LIN {X 0,Y 523.995,Z 483.842,A -85,B 0,C 180,E1 -4869.262,E2 -4869.262} C_VEL
LIN {X 0,Y 523.998,Z 483.841,A -85,B 0,C 180,E1 -4871.743,E2 -4871.743} C_VEL
LIN {X 0,Y 523.983,Z 483.844,A -85,B 0,C 180,E1 -4875.053,E2 -4875.053} C_VEL
LIN {X 0,Y 523.956,Z 483.847,A -85,B 0,C 180,E1 -4877.97,E2 -4877.97} C_VEL
LIN {X 0,Y 523.964,Z 483.845,A -85,B 0,C 180,E1 -4880.411,E2 -4880.411} C_VEL
LIN {X 0,Y 523.909,Z 483.852,A -85,B 0,C 180,E1 -4882.894,E2 -4882.894} C_VEL
LIN {X 0,Y 523.947,Z 483.847,A -85,B 0,C 180,E1 -4885.419,E2 -4885.419} C_VEL
LIN {X 0,Y 523.964,Z 483.846,A -85,B 0,C 180,E1 -4888,E2 -4888} C_VEL
LIN {X 0,Y 523.946,Z 483.846,A -85,B 0,C 180,E1 -4890.857,E2 -4890.857} C_VEL
LIN {X 0,Y 523.957,Z 483.847,A -85,B 0,C 180,E1 -4893.736,E2 -4893.736} C_VEL
LIN {X 0,Y 523.917,Z 483.849,A -85,B 0,C 180,E1 -4896.405,E2 -4896.405} C_VEL
LIN {X 0,Y 523.956,Z 483.846,A -85,B 0,C 180,E1 -4899.082,E2 -4899.082} C_VEL
LIN {X 0,Y 523.962,Z 483.845,A -85,B 0,C 180,E1 -4902.119,E2 -4902.119} C_VEL
LIN {X 0,Y 523.953,Z 483.846,A -85,B 0,C 180,E1 -4905.31,E2 -4905.31} C_VEL
LIN {X 0,Y 523.92,Z 483.85,A -85,B 0,C 180,E1 -4906.926,E2 -4906.926} C_VEL
LIN {X 0,Y 523.256,Z 483.934,A -85,B 0,C 180,E1 -4907.567,E2 -4907.567} C_VEL
LIN {X 0,Y 520.42,Z 484.287,A -85,B 0,C 180,E1 -4908.609,E2 -4908.609} C_VEL
LIN {X 0,Y 518.024,Z 484.586,A -85,B 0,C 180,E1 -4909.449,E2 -4909.449} C_VEL
LIN {X 0,Y 516.994,Z 484.714,A -85,B 0,C 180,E1 -4910.096,E2 -4910.096} C_VEL
LIN {X 0,Y 516.909,Z 484.722,A -85,B 0,C 180,E1 -4910.316,E2 -4910.316} C_VEL
LIN {X 0,Y 516.884,Z 484.728,A -85,B 0,C 180,E1 -4913.343,E2 -4913.343} C_VEL
LIN {X 0,Y 516.911,Z 484.723,A -85,B 0,C 180,E1 -4916.122,E2 -4916.122} C_VEL
LIN {X 0,Y 516.893,Z 484.726,A -85,B 0,C 180,E1 -4918.936,E2 -4918.936} C_VEL
LIN {X 0,Y 516.922,Z 484.722,A -85,B 0,C 180,E1 -4921.586,E2 -4921.586} C_VEL
LIN {X 0,Y 516.936,Z 484.721,A -85,B 0,C 180,E1 -4924.212,E2 -4924.212} C_VEL
LIN {X 0,Y 516.875,Z 484.728,A -85,B 0,C 180,E1 -4926.778,E2 -4926.778} C_VEL
LIN {X 0,Y 516.942,Z 484.72,A -85,B 0,C 180,E1 -4929.733,E2 -4929.733} C_VEL
LIN {X 0,Y 516.933,Z 484.719,A -85,B 0,C 180,E1 -4932.597,E2 -4932.597} C_VEL
LIN {X 0,Y 516.947,Z 484.718,A -85,B 0,C 180,E1 -4935.031,E2 -4935.031} C_VEL
LIN {X 0,Y 516.971,Z 484.715,A -85,B 0,C 180,E1 -4938.234,E2 -4938.234} C_VEL
LIN {X 0,Y 516.961,Z 484.717,A -85,B 0,C 180,E1 -4941.4,E2 -4941.4} C_VEL
LIN {X 0,Y 517.016,Z 484.71,A -85,B 0,C 180,E1 -4943.757,E2 -4943.757} C_VEL
LIN {X 0,Y 517.09,Z 484.703,A -85,B 0,C 180,E1 -4947.664,E2 -4947.664} C_VEL
LIN {X 0,Y 517.098,Z 484.699,A -85,B 0,C 180,E1 -4950.779,E2 -4950.779} C_VEL
LIN {X 0,Y 517.003,Z 484.713,A -85,B 0,C 180,E1 -4952.338,E2 -4952.338} C_VEL
LIN {X 0,Y 516.745,Z 484.747,A -85,B 0,C 180,E1 -4954.681,E2 -4954.681} C_VEL
LIN {X 0,Y 516.605,Z 485.864,A -85,B 0,C 180,E1 -4956.248,E2 -4956.248} C_VEL
LIN {X 0,Y 516.544,Z 488.063,A -85,B 0,C 180,E1 -4958.608,E2 -4958.608} C_VEL
LIN {X 0,Y 516.481,Z 491.026,A -85,B 0,C 180,E1 -4961.778,E2 -4961.778} C_VEL
LIN {X 0,Y 516.458,Z 493.998,A -85,B 0,C 180,E1 -4964.984,E2 -4964.984} C_VEL
LIN {X 0,Y 516.325,Z 497.059,A -85,B 0,C 180,E1 -4968.244,E2 -4968.244} C_VEL
LIN {X 0,Y 516.284,Z 499.09,A -85,B 0,C 180,E1 -4970.448,E2 -4970.448} C_VEL
LIN {X 0,Y 520.67,Z 515.911,A -85,B 0,C 180,E1 -4970.996,E2 -4970.996} C_VEL
LIN {X 0,Y 520.325,Z 530.084,A -85,B 0,C 180,E1 -4971.44,E2 -4971.44} C_VEL
LIN {X 0,Y 519.941,Z 544.068,A -85,B 0,C 180,E1 -4972.03,E2 -4972.03} C_VEL
LIN {X 0,Y 519.433,Z 557.792,A -85,B 0,C 180,E1 -4972.767,E2 -4972.767} C_VEL
LIN {X 0,Y 518.868,Z 571.154,A -85,B 0,C 180,E1 -4973.657,E2 -4973.657} C_VEL
LIN {X 0,Y 518.342,Z 584.059,A -85,B 0,C 180,E1 -4974.71,E2 -4974.71} C_VEL
LIN {X 0,Y 517.781,Z 596.388,A -85,B 0,C 180,E1 -4975.926,E2 -4975.926} C_VEL
LIN {X 0,Y 517.395,Z 606.182,A -85,B 0,C 180,E1 -4977.068,E2 -4977.068} C_VEL
LIN {X 0,Y 517.038,Z 615.882,A -85,B 0,C 180,E1 -4978.408,E2 -4978.408} C_VEL
LIN {X 0,Y 516.758,Z 624.427,A -85,B 0,C 180,E1 -4979.823,E2 -4979.823} C_VEL
LIN {X 0,Y 516.533,Z 632.07,A -85,B 0,C 180,E1 -4981.361,E2 -4981.361} C_VEL
LIN {X 0,Y 516.343,Z 638.529,A -85,B 0,C 180,E1 -4982.986,E2 -4982.986} C_VEL
LIN {X 0,Y 516.285,Z 642.897,A -85,B 0,C 180,E1 -4984.397,E2 -4984.397} C_VEL
LIN {X 0,Y 516.177,Z 646.315,A -85,B 0,C 180,E1 -4985.836,E2 -4985.836} C_VEL
LIN {X 0,Y 516.137,Z 648.013,A -85,B 0,C 180,E1 -4986.807,E2 -4986.807} C_VEL
LIN {X 0,Y 516.138,Z 649.321,A -85,B 0,C 180,E1 -4987.836,E2 -4987.836} C_VEL
LIN {X 0,Y 516.128,Z 650.278,A -85,B 0,C 180,E1 -4989.089,E2 -4989.089} C_VEL
LIN {X 0,Y 516.139,Z 650.35,A -85,B 0,C 180,E1 -4990.812,E2 -4990.812} C_VEL
LIN {X 0,Y 516.146,Z 649.734,A -85,B 0,C 180,E1 -4991.851,E2 -4991.851} C_VEL
LIN {X 0,Y 516.173,Z 648.562,A -85,B 0,C 180,E1 -4992.904,E2 -4992.904} C_VEL
LIN {X 0,Y 516.264,Z 645.924,A -85,B 0,C 180,E1 -4994.452,E2 -4994.452} C_VEL
LIN {X 0,Y 516.317,Z 641.557,A -85,B 0,C 180,E1 -4996.172,E2 -4996.172} C_VEL
LIN {X 0,Y 516.429,Z 636.204,A -85,B 0,C 180,E1 -4997.742,E2 -4997.742} C_VEL
LIN {X 0,Y 516.543,Z 629.799,A -85,B 0,C 180,E1 -4999.225,E2 -4999.225} C_VEL
LIN {X 0,Y 516.833,Z 621.343,A -85,B 0,C 180,E1 -5000.813,E2 -5000.813} C_VEL
LIN {X 0,Y 517.202,Z 611.617,A -85,B 0,C 180,E1 -5002.303,E2 -5002.303} C_VEL
LIN {X 0,Y 517.602,Z 600.766,A -85,B 0,C 180,E1 -5003.676,E2 -5003.676} C_VEL
LIN {X 0,Y 518.126,Z 589.032,A -85,B 0,C 180,E1 -5004.915,E2 -5004.915} C_VEL
LIN {X 0,Y 518.638,Z 576.91,A -85,B 0,C 180,E1 -5005.988,E2 -5005.988} C_VEL
LIN {X 0,Y 519.165,Z 563.866,A -85,B 0,C 180,E1 -5006.944,E2 -5006.944} C_VEL
LIN {X 0,Y 519.71,Z 549.92,A -85,B 0,C 180,E1 -5007.77,E2 -5007.77} C_VEL
LIN {X 0,Y 520.223,Z 535.183,A -85,B 0,C 180,E1 -5008.455,E2 -5008.455} C_VEL
LIN {X 0,Y 520.534,Z 520.831,A -85,B 0,C 180,E1 -5008.963,E2 -5008.963} C_VEL
LIN {X 0,Y 520.482,Z 515.011,A -85,B 0,C 180,E1 -5009.128,E2 -5009.128} C_VEL
LIN {X 0,Y 517.023,Z 501.814,A -85,B 0,C 180,E1 -5009.551,E2 -5009.551} C_VEL
LIN {X 0,Y 516.31,Z 499.259,A -85,B 0,C 180,E1 -5009.646,E2 -5009.646} C_VEL
LIN {X 0,Y 516.359,Z 496.719,A -85,B 0,C 180,E1 -5012.434,E2 -5012.434} C_VEL
LIN {X 0,Y 516.419,Z 494.464,A -85,B 0,C 180,E1 -5015.046,E2 -5015.046} C_VEL
LIN {X 0,Y 516.472,Z 492.208,A -85,B 0,C 180,E1 -5017.716,E2 -5017.716} C_VEL
LIN {X 0,Y 516.573,Z 490.1,A -85,B 0,C 180,E1 -5020.115,E2 -5020.115} C_VEL
LIN {X 0,Y 516.622,Z 487.924,A -85,B 0,C 180,E1 -5022.585,E2 -5022.585} C_VEL
LIN {X 0,Y 516.669,Z 485.071,A -85,B 0,C 180,E1 -5025.827,E2 -5025.827} C_VEL
LIN {X 0,Y 516.789,Z 484.742,A -85,B 0,C 180,E1 -5027.432,E2 -5027.432} C_VEL
LIN {X 0,Y 516.904,Z 484.725,A -85,B 0,C 180,E1 -5029.819,E2 -5029.819} C_VEL
LIN {X 0,Y 516.976,Z 484.716,A -85,B 0,C 180,E1 -5032.186,E2 -5032.186} C_VEL
LIN {X 0,Y 517.032,Z 484.704,A -85,B 0,C 180,E1 -5034.54,E2 -5034.54} C_VEL
LIN {X 0,Y 517.081,Z 484.704,A -85,B 0,C 180,E1 -5037.663,E2 -5037.663} C_VEL
LIN {X 0,Y 517.091,Z 484.696,A -85,B 0,C 180,E1 -5040.778,E2 -5040.778} C_VEL
LIN {X 0,Y 517.011,Z 484.71,A -85,B 0,C 180,E1 -5043.117,E2 -5043.117} C_VEL
LIN {X 0,Y 517.007,Z 484.706,A -85,B 0,C 180,E1 -5046.243,E2 -5046.243} C_VEL
LIN {X 0,Y 516.952,Z 484.717,A -85,B 0,C 180,E1 -5049.389,E2 -5049.389} C_VEL
LIN {X 0,Y 516.953,Z 484.713,A -85,B 0,C 180,E1 -5051.81,E2 -5051.81} C_VEL
LIN {X 0,Y 516.94,Z 484.717,A -85,B 0,C 180,E1 -5055.146,E2 -5055.146} C_VEL
LIN {X 0,Y 516.921,Z 484.719,A -85,B 0,C 180,E1 -5058.222,E2 -5058.222} C_VEL
LIN {X 0,Y 516.909,Z 484.723,A -85,B 0,C 180,E1 -5060.701,E2 -5060.701} C_VEL
LIN {X 0,Y 516.907,Z 484.723,A -85,B 0,C 180,E1 -5064.072,E2 -5064.072} C_VEL
LIN {X 0,Y 516.925,Z 484.719,A -85,B 0,C 180,E1 -5066.658,E2 -5066.658} C_VEL
LIN {X 0,Y 516.921,Z 484.72,A -85,B 0,C 180,E1 -5069.527,E2 -5069.527} C_VEL
LIN {X 0,Y 516.897,Z 484.721,A -85,B 0,C 180,E1 -5072.544,E2 -5072.544} C_VEL
LIN {X 0,Y 516.88,Z 484.726,A -85,B 0,C 180,E1 -5075.333,E2 -5075.333} C_VEL
LIN {X 0,Y 516.879,Z 484.725,A -85,B 0,C 180,E1 -5077.943,E2 -5077.943} C_VEL
LIN {X 0,Y 516.883,Z 484.723,A -85,B 0,C 180,E1 -5080.741,E2 -5080.741} C_VEL
LIN {X 0,Y 516.902,Z 484.725,A -85,B 0,C 180,E1 -5082.829,E2 -5082.829} C_VEL
LIN {X 0,Y 516.941,Z 484.824,A -85,B 0,C 180,E1 -5084.85,E2 -5084.85} C_VEL
LIN {X 0,Y 517.947,Z 490.869,A -85,B 0,C 180,E1 -5087.805,E2 -5087.805} C_VEL
LIN {X 0,Y 518.047,Z 495.695,A -85,B 0,C 180,E1 -5089.911,E2 -5089.911} C_VEL
LIN {X 0,Y 517.767,Z 502.856,A -85,B 0,C 180,E1 -5092.828,E2 -5092.828} C_VEL
LIN {X 0,Y 517.6,Z 509.05,A -85,B 0,C 180,E1 -5095.231,E2 -5095.231} C_VEL
LIN {X 0,Y 517.428,Z 517.921,A -85,B 0,C 180,E1 -5098.472,E2 -5098.472} C_VEL
LIN {X 0,Y 517.211,Z 526.908,A -85,B 0,C 180,E1 -5101.602,E2 -5101.602} C_VEL
LIN {X 0,Y 517.044,Z 535.926,A -85,B 0,C 180,E1 -5104.649,E2 -5104.649} C_VEL
LIN {X 0,Y 516.914,Z 545.207,A -85,B 0,C 180,E1 -5107.624,E2 -5107.624} C_VEL
LIN {X 0,Y 516.827,Z 554.056,A -85,B 0,C 180,E1 -5110.384,E2 -5110.384} C_VEL
LIN {X 0,Y 520.741,Z 570.926,A -85,B 0,C 180,E1 -5110.845,E2 -5110.845} C_VEL
LIN {X 0,Y 520.347,Z 586.426,A -85,B 0,C 180,E1 -5111.287,E2 -5111.287} C_VEL
LIN {X 0,Y 519.937,Z 601.506,A -85,B 0,C 180,E1 -5111.887,E2 -5111.887} C_VEL
LIN {X 0,Y 519.531,Z 615.077,A -85,B 0,C 180,E1 -5112.584,E2 -5112.584} C_VEL
LIN {X 0,Y 519.01,Z 627.615,A -85,B 0,C 180,E1 -5113.378,E2 -5113.378} C_VEL
LIN {X 0,Y 518.491,Z 640.647,A -85,B 0,C 180,E1 -5114.382,E2 -5114.382} C_VEL
LIN {X 0,Y 517.981,Z 652.324,A -85,B 0,C 180,E1 -5115.463,E2 -5115.463} C_VEL
LIN {X 0,Y 517.552,Z 663.136,A -85,B 0,C 180,E1 -5116.653,E2 -5116.653} C_VEL
LIN {X 0,Y 517.081,Z 673.797,A -85,B 0,C 180,E1 -5118.057,E2 -5118.057} C_VEL
LIN {X 0,Y 516.89,Z 682.414,A -85,B 0,C 180,E1 -5119.423,E2 -5119.423} C_VEL
LIN {X 0,Y 516.638,Z 688.748,A -85,B 0,C 180,E1 -5120.605,E2 -5120.605} C_VEL
LIN {X 0,Y 516.463,Z 695.699,A -85,B 0,C 180,E1 -5122.179,E2 -5122.179} C_VEL
LIN {X 0,Y 516.356,Z 701.161,A -85,B 0,C 180,E1 -5123.749,E2 -5123.749} C_VEL
LIN {X 0,Y 516.239,Z 705.29,A -85,B 0,C 180,E1 -5125.314,E2 -5125.314} C_VEL
LIN {X 0,Y 516.272,Z 708.184,A -85,B 0,C 180,E1 -5126.878,E2 -5126.878} C_VEL
LIN {X 0,Y 516.189,Z 709.909,A -85,B 0,C 180,E1 -5128.439,E2 -5128.439} C_VEL
LIN {X 0,Y 516.151,Z 710.5,A -85,B 0,C 180,E1 -5130,E2 -5130} C_VEL
LIN {X 0,Y 516.189,Z 709.907,A -85,B 0,C 180,E1 -5131.56,E2 -5131.56} C_VEL
LIN {X 0,Y 516.272,Z 708.181,A -85,B 0,C 180,E1 -5133.121,E2 -5133.121} C_VEL
LIN {X 0,Y 516.238,Z 705.289,A -85,B 0,C 180,E1 -5134.685,E2 -5134.685} C_VEL
LIN {X 0,Y 516.349,Z 701.167,A -85,B 0,C 180,E1 -5136.251,E2 -5136.251} C_VEL
LIN {X 0,Y 516.462,Z 695.703,A -85,B 0,C 180,E1 -5137.821,E2 -5137.821} C_VEL
LIN {X 0,Y 516.637,Z 688.746,A -85,B 0,C 180,E1 -5139.394,E2 -5139.394} C_VEL
LIN {X 0,Y 516.971,Z 680.085,A -85,B 0,C 180,E1 -5140.971,E2 -5140.971} C_VEL
LIN {X 0,Y 517.224,Z 671.026,A -85,B 0,C 180,E1 -5142.337,E2 -5142.337} C_VEL
LIN {X 0,Y 517.633,Z 661.513,A -85,B 0,C 180,E1 -5143.544,E2 -5143.544} C_VEL
LIN {X 0,Y 518.114,Z 649.368,A -85,B 0,C 180,E1 -5144.834,E2 -5144.834} C_VEL
LIN {X 0,Y 518.624,Z 637.232,A -85,B 0,C 180,E1 -5145.906,E2 -5145.906} C_VEL
LIN {X 0,Y 519.093,Z 624.775,A -85,B 0,C 180,E1 -5146.821,E2 -5146.821} C_VEL
LIN {X 0,Y 519.647,Z 611.528,A -85,B 0,C 180,E1 -5147.614,E2 -5147.614} C_VEL
LIN {X 0,Y 520.055,Z 598.266,A -85,B 0,C 180,E1 -5148.255,E2 -5148.255} C_VEL
LIN {X 0,Y 520.479,Z 583.266,A -85,B 0,C 180,E1 -5148.816,E2 -5148.816} C_VEL
LIN {X 0,Y 520.641,Z 570.407,A -85,B 0,C 180,E1 -5149.172,E2 -5149.172} C_VEL
LIN {X 0,Y 516.816,Z 554.06,A -85,B 0,C 180,E1 -5149.622,E2 -5149.622} C_VEL
LIN {X 0,Y 516.973,Z 544.246,A -85,B 0,C 180,E1 -5152.794,E2 -5152.794} C_VEL
LIN {X 0,Y 517.135,Z 535.156,A -85,B 0,C 180,E1 -5155.777,E2 -5155.777} C_VEL
LIN {X 0,Y 517.291,Z 526.189,A -85,B 0,C 180,E1 -5158.835,E2 -5158.835} C_VEL
LIN {X 0,Y 517.499,Z 518.635,A -85,B 0,C 180,E1 -5161.529,E2 -5161.529} C_VEL
LIN {X 0,Y 517.644,Z 511.67,A -85,B 0,C 180,E1 -5164.087,E2 -5164.087} C_VEL
LIN {X 0,Y 517.876,Z 503.58,A -85,B 0,C 180,E1 -5167.176,E2 -5167.176} C_VEL
LIN {X 0,Y 518.18,Z 496.323,A -85,B 0,C 180,E1 -5170.093,E2 -5170.093} C_VEL
LIN {X 0,Y 518.175,Z 492.369,A -85,B 0,C 180,E1 -5171.758,E2 -5171.758} C_VEL
LIN {X 0,Y 517.405,Z 487.511,A -85,B 0,C 180,E1 -5173.953,E2 -5173.953} C_VEL
LIN {X 0,Y 516.928,Z 484.72,A -85,B 0,C 180,E1 -5175.285,E2 -5175.285} C_VEL
LIN {X 0,Y 516.922,Z 484.722,A -85,B 0,C 180,E1 -5178.396,E2 -5178.396} C_VEL
LIN {X 0,Y 516.899,Z 484.725,A -85,B 0,C 180,E1 -5181.286,E2 -5181.286} C_VEL
LIN {X 0,Y 516.883,Z 484.727,A -85,B 0,C 180,E1 -5184.221,E2 -5184.221} C_VEL
LIN {X 0,Y 516.89,Z 484.725,A -85,B 0,C 180,E1 -5187.053,E2 -5187.053} C_VEL
LIN {X 0,Y 516.893,Z 484.726,A -85,B 0,C 180,E1 -5189.797,E2 -5189.797} C_VEL
LIN {X 0,Y 516.921,Z 484.72,A -85,B 0,C 180,E1 -5192.467,E2 -5192.467} C_VEL
LIN {X 0,Y 516.902,Z 484.724,A -85,B 0,C 180,E1 -5195.072,E2 -5195.072} C_VEL
LIN {X 0,Y 516.877,Z 484.727,A -85,B 0,C 180,E1 -5198.462,E2 -5198.462} C_VEL
LIN {X 0,Y 516.896,Z 484.726,A -85,B 0,C 180,E1 -5200.955,E2 -5200.955} C_VEL
LIN {X 0,Y 516.908,Z 484.724,A -85,B 0,C 180,E1 -5203.41,E2 -5203.41} C_VEL
LIN {X 0,Y 516.885,Z 484.727,A -85,B 0,C 180,E1 -5205.834,E2 -5205.834} C_VEL
LIN {X 0,Y 516.993,Z 484.714,A -85,B 0,C 180,E1 -5208.235,E2 -5208.235} C_VEL
LIN {X 0,Y 516.964,Z 484.717,A -85,B 0,C 180,E1 -5211.4,E2 -5211.4} C_VEL
LIN {X 0,Y 517.036,Z 484.705,A -85,B 0,C 180,E1 -5214.54,E2 -5214.54} C_VEL
LIN {X 0,Y 517.076,Z 484.703,A -85,B 0,C 180,E1 -5217.663,E2 -5217.663} C_VEL
LIN {X 0,Y 517.086,Z 484.702,A -85,B 0,C 180,E1 -5220.779,E2 -5220.779} C_VEL
LIN {X 0,Y 517.01,Z 484.711,A -85,B 0,C 180,E1 -5223.117,E2 -5223.117} C_VEL
LIN {X 0,Y 517.007,Z 484.71,A -85,B 0,C 180,E1 -5226.244,E2 -5226.244} C_VEL
LIN {X 0,Y 516.949,Z 484.72,A -85,B 0,C 180,E1 -5229.39,E2 -5229.39} C_VEL
LIN {X 0,Y 516.947,Z 484.719,A -85,B 0,C 180,E1 -5231.811,E2 -5231.811} C_VEL
LIN {X 0,Y 516.934,Z 484.721,A -85,B 0,C 180,E1 -5235.147,E2 -5235.147} C_VEL
LIN {X 0,Y 516.917,Z 484.722,A -85,B 0,C 180,E1 -5238.223,E2 -5238.223} C_VEL
LIN {X 0,Y 516.904,Z 484.724,A -85,B 0,C 180,E1 -5240.702,E2 -5240.702} C_VEL
LIN {X 0,Y 516.903,Z 484.723,A -85,B 0,C 180,E1 -5244.073,E2 -5244.073} C_VEL
LIN {X 0,Y 516.923,Z 484.72,A -85,B 0,C 180,E1 -5246.658,E2 -5246.658} C_VEL
LIN {X 0,Y 516.918,Z 484.723,A -85,B 0,C 180,E1 -5249.528,E2 -5249.528} C_VEL
LIN {X 0,Y 516.895,Z 484.725,A -85,B 0,C 180,E1 -5252.546,E2 -5252.546} C_VEL
LIN {X 0,Y 516.878,Z 484.727,A -85,B 0,C 180,E1 -5255.334,E2 -5255.334} C_VEL
LIN {X 0,Y 516.877,Z 484.729,A -85,B 0,C 180,E1 -5257.945,E2 -5257.945} C_VEL
LIN {X 0,Y 516.913,Z 484.721,A -85,B 0,C 180,E1 -5260.739,E2 -5260.739} C_VEL
LIN {X 0,Y 516.879,Z 484.727,A -85,B 0,C 180,E1 -5263.904,E2 -5263.904} C_VEL
LIN {X 0,Y 516.879,Z 484.726,A -85,B 0,C 180,E1 -5266.108,E2 -5266.108} C_VEL
LIN {X 0,Y 516.903,Z 484.725,A -85,B 0,C 180,E1 -5269.262,E2 -5269.262} C_VEL
LIN {X 0,Y 516.909,Z 484.722,A -85,B 0,C 180,E1 -5270.316,E2 -5270.316} C_VEL
LIN {X 0,Y 516.24,Z 484.806,A -85,B 0,C 180,E1 -5270.966,E2 -5270.966} C_VEL
LIN {X 0,Y 513.383,Z 485.163,A -85,B 0,C 180,E1 -5272.021,E2 -5272.021} C_VEL
LIN {X 0,Y 510.964,Z 485.467,A -85,B 0,C 180,E1 -5272.871,E2 -5272.871} C_VEL
LIN {X 0,Y 509.918,Z 485.596,A -85,B 0,C 180,E1 -5273.527,E2 -5273.527} C_VEL
LIN {X 0,Y 509.829,Z 485.605,A -85,B 0,C 180,E1 -5273.75,E2 -5273.75} C_VEL
LIN {X 0,Y 509.861,Z 485.601,A -85,B 0,C 180,E1 -5276.54,E2 -5276.54} C_VEL
LIN {X 0,Y 509.847,Z 485.604,A -85,B 0,C 180,E1 -5279.335,E2 -5279.335} C_VEL
LIN {X 0,Y 509.897,Z 485.598,A -85,B 0,C 180,E1 -5282.056,E2 -5282.056} C_VEL
LIN {X 0,Y 509.881,Z 485.598,A -85,B 0,C 180,E1 -5284.705,E2 -5284.705} C_VEL
LIN {X 0,Y 509.839,Z 485.604,A -85,B 0,C 180,E1 -5287.456,E2 -5287.456} C_VEL
LIN {X 0,Y 509.92,Z 485.596,A -85,B 0,C 180,E1 -5289.846,E2 -5289.846} C_VEL
LIN {X 0,Y 509.889,Z 485.598,A -85,B 0,C 180,E1 -5293.176,E2 -5293.176} C_VEL
LIN {X 0,Y 509.868,Z 485.602,A -85,B 0,C 180,E1 -5295.635,E2 -5295.635} C_VEL
LIN {X 0,Y 509.917,Z 485.594,A -85,B 0,C 180,E1 -5298.875,E2 -5298.875} C_VEL
LIN {X 0,Y 509.926,Z 485.594,A -85,B 0,C 180,E1 -5302.079,E2 -5302.079} C_VEL
LIN {X 0,Y 509.987,Z 485.585,A -85,B 0,C 180,E1 -5304.465,E2 -5304.465} C_VEL
LIN {X 0,Y 510.061,Z 485.578,A -85,B 0,C 180,E1 -5307.631,E2 -5307.631} C_VEL
LIN {X 0,Y 510.069,Z 485.575,A -85,B 0,C 180,E1 -5310.79,E2 -5310.79} C_VEL
LIN {X 0,Y 509.943,Z 485.592,A -85,B 0,C 180,E1 -5312.37,E2 -5312.37} C_VEL
LIN {X 0,Y 509.702,Z 485.624,A -85,B 0,C 180,E1 -5314.746,E2 -5314.746} C_VEL
LIN {X 0,Y 509.527,Z 485.909,A -85,B 0,C 180,E1 -5315.541,E2 -5315.541} C_VEL
LIN {X 0,Y 509.505,Z 488.136,A -85,B 0,C 180,E1 -5317.929,E2 -5317.929} C_VEL
LIN {X 0,Y 509.419,Z 491.088,A -85,B 0,C 180,E1 -5321.137,E2 -5321.137} C_VEL
LIN {X 0,Y 509.387,Z 494.091,A -85,B 0,C 180,E1 -5324.38,E2 -5324.38} C_VEL
LIN {X 0,Y 509.289,Z 497.265,A -85,B 0,C 180,E1 -5327.79,E2 -5327.79} C_VEL
LIN {X 0,Y 509.245,Z 499.51,A -85,B 0,C 180,E1 -5330.183,E2 -5330.183} C_VEL
LIN {X 0,Y 513.235,Z 514.056,A -85,B 0,C 180,E1 -5330.647,E2 -5330.647} C_VEL
LIN {X 0,Y 513.945,Z 517.527,A -85,B 0,C 180,E1 -5330.774,E2 -5330.774} C_VEL
LIN {X 0,Y 513.583,Z 531.701,A -85,B 0,C 180,E1 -5331.239,E2 -5331.239} C_VEL
LIN {X 0,Y 513.135,Z 545.901,A -85,B 0,C 180,E1 -5331.862,E2 -5331.862} C_VEL
LIN {X 0,Y 512.643,Z 558.776,A -85,B 0,C 180,E1 -5332.573,E2 -5332.573} C_VEL
LIN {X 0,Y 512.032,Z 571.804,A -85,B 0,C 180,E1 -5333.456,E2 -5333.456} C_VEL
LIN {X 0,Y 511.472,Z 584.438,A -85,B 0,C 180,E1 -5334.501,E2 -5334.501} C_VEL
LIN {X 0,Y 510.913,Z 596.247,A -85,B 0,C 180,E1 -5335.677,E2 -5335.677} C_VEL
LIN {X 0,Y 510.384,Z 607.493,A -85,B 0,C 180,E1 -5337.027,E2 -5337.027} C_VEL
LIN {X 0,Y 509.977,Z 617.324,A -85,B 0,C 180,E1 -5338.45,E2 -5338.45} C_VEL
LIN {X 0,Y 509.664,Z 626.083,A -85,B 0,C 180,E1 -5339.991,E2 -5339.991} C_VEL
LIN {X 0,Y 509.459,Z 631.923,A -85,B 0,C 180,E1 -5341.207,E2 -5341.207} C_VEL
LIN {X 0,Y 509.279,Z 637.747,A -85,B 0,C 180,E1 -5342.669,E2 -5342.669} C_VEL
LIN {X 0,Y 509.201,Z 642.294,A -85,B 0,C 180,E1 -5344.093,E2 -5344.093} C_VEL
LIN {X 0,Y 509.092,Z 645.666,A -85,B 0,C 180,E1 -5345.462,E2 -5345.462} C_VEL
LIN {X 0,Y 509.042,Z 648.06,A -85,B 0,C 180,E1 -5346.796,E2 -5346.796} C_VEL
LIN {X 0,Y 509.037,Z 649.874,A -85,B 0,C 180,E1 -5348.41,E2 -5348.41} C_VEL
LIN {X 0,Y 509.028,Z 650.382,A -85,B 0,C 180,E1 -5349.428,E2 -5349.428} C_VEL
LIN {X 0,Y 509.051,Z 650.396,A -85,B 0,C 180,E1 -5350.594,E2 -5350.594} C_VEL
LIN {X 0,Y 509.044,Z 649.806,A -85,B 0,C 180,E1 -5351.794,E2 -5351.794} C_VEL
LIN {X 0,Y 509.103,Z 647.535,A -85,B 0,C 180,E1 -5353.648,E2 -5353.648} C_VEL
LIN {X 0,Y 509.195,Z 644.248,A -85,B 0,C 180,E1 -5355.258,E2 -5355.258} C_VEL
LIN {X 0,Y 509.295,Z 639.231,A -85,B 0,C 180,E1 -5357.001,E2 -5357.001} C_VEL
LIN {X 0,Y 509.38,Z 633.476,A -85,B 0,C 180,E1 -5358.527,E2 -5358.527} C_VEL
LIN {X 0,Y 509.652,Z 626.075,A -85,B 0,C 180,E1 -5360.103,E2 -5360.103} C_VEL
LIN {X 0,Y 509.969,Z 617.151,A -85,B 0,C 180,E1 -5361.672,E2 -5361.672} C_VEL
LIN {X 0,Y 510.371,Z 607.96,A -85,B 0,C 180,E1 -5363.004,E2 -5363.004} C_VEL
LIN {X 0,Y 510.904,Z 596.892,A -85,B 0,C 180,E1 -5364.345,E2 -5364.345} C_VEL
LIN {X 0,Y 511.493,Z 585.133,A -85,B 0,C 180,E1 -5365.528,E2 -5365.528} C_VEL
LIN {X 0,Y 512.029,Z 572.556,A -85,B 0,C 180,E1 -5366.581,E2 -5366.581} C_VEL
LIN {X 0,Y 512.573,Z 560.098,A -85,B 0,C 180,E1 -5367.441,E2 -5367.441} C_VEL
LIN {X 0,Y 513.024,Z 547.804,A -85,B 0,C 180,E1 -5368.14,E2 -5368.14} C_VEL
LIN {X 0,Y 513.533,Z 533.681,A -85,B 0,C 180,E1 -5368.778,E2 -5368.778} C_VEL
LIN {X 0,Y 513.915,Z 519.1,A -85,B 0,C 180,E1 -5369.275,E2 -5369.275} C_VEL
LIN {X 0,Y 513.625,Z 515.708,A -85,B 0,C 180,E1 -5369.384,E2 -5369.384} C_VEL
LIN {X 0,Y 510.164,Z 502.851,A -85,B 0,C 180,E1 -5369.813,E2 -5369.813} C_VEL
LIN {X 0,Y 509.276,Z 499.766,A -85,B 0,C 180,E1 -5369.926,E2 -5369.926} C_VEL
LIN {X 0,Y 509.289,Z 497.11,A -85,B 0,C 180,E1 -5372.91,E2 -5372.91} C_VEL
LIN {X 0,Y 509.377,Z 494.831,A -85,B 0,C 180,E1 -5375.59,E2 -5375.59} C_VEL
LIN {X 0,Y 509.42,Z 492.583,A -85,B 0,C 180,E1 -5378.13,E2 -5378.13} C_VEL
LIN {X 0,Y 509.496,Z 490.376,A -85,B 0,C 180,E1 -5380.667,E2 -5380.667} C_VEL
LIN {X 0,Y 509.544,Z 488.22,A -85,B 0,C 180,E1 -5383.163,E2 -5383.163} C_VEL
LIN {X 0,Y 509.626,Z 486.077,A -85,B 0,C 180,E1 -5385.627,E2 -5385.627} C_VEL
LIN {X 0,Y 509.642,Z 485.631,A -85,B 0,C 180,E1 -5386.442,E2 -5386.442} C_VEL
LIN {X 0,Y 509.89,Z 485.596,A -85,B 0,C 180,E1 -5388.874,E2 -5388.874} C_VEL
LIN {X 0,Y 509.949,Z 485.592,A -85,B 0,C 180,E1 -5392.078,E2 -5392.078} C_VEL
LIN {X 0,Y 509.983,Z 485.583,A -85,B 0,C 180,E1 -5394.464,E2 -5394.464} C_VEL
LIN {X 0,Y 510.052,Z 485.579,A -85,B 0,C 180,E1 -5397.631,E2 -5397.631} C_VEL
LIN {X 0,Y 510.061,Z 485.572,A -85,B 0,C 180,E1 -5400.789,E2 -5400.789} C_VEL
LIN {X 0,Y 509.953,Z 485.59,A -85,B 0,C 180,E1 -5403.16,E2 -5403.16} C_VEL
LIN {X 0,Y 509.975,Z 485.582,A -85,B 0,C 180,E1 -5406.329,E2 -5406.329} C_VEL
LIN {X 0,Y 509.913,Z 485.593,A -85,B 0,C 180,E1 -5408.72,E2 -5408.72} C_VEL
LIN {X 0,Y 509.901,Z 485.591,A -85,B 0,C 180,E1 -5411.931,E2 -5411.931} C_VEL
LIN {X 0,Y 509.889,Z 485.595,A -85,B 0,C 180,E1 -5415.242,E2 -5415.242} C_VEL
LIN {X 0,Y 509.884,Z 485.594,A -85,B 0,C 180,E1 -5418.001,E2 -5418.001} C_VEL
LIN {X 0,Y 509.847,Z 485.599,A -85,B 0,C 180,E1 -5421.002,E2 -5421.002} C_VEL
LIN {X 0,Y 509.833,Z 485.599,A -85,B 0,C 180,E1 -5423.563,E2 -5423.563} C_VEL
LIN {X 0,Y 509.91,Z 485.595,A -85,B 0,C 180,E1 -5426.379,E2 -5426.379} C_VEL
LIN {X 0,Y 509.882,Z 485.595,A -85,B 0,C 180,E1 -5428.844,E2 -5428.844} C_VEL
LIN {X 0,Y 509.824,Z 485.606,A -85,B 0,C 180,E1 -5431.59,E2 -5431.59} C_VEL
LIN {X 0,Y 509.851,Z 485.599,A -85,B 0,C 180,E1 -5434.413,E2 -5434.413} C_VEL
LIN {X 0,Y 509.816,Z 485.607,A -85,B 0,C 180,E1 -5437.341,E2 -5437.341} C_VEL
LIN {X 0,Y 509.836,Z 485.6,A -85,B 0,C 180,E1 -5440.382,E2 -5440.382} C_VEL
LIN {X 0,Y 509.837,Z 485.606,A -85,B 0,C 180,E1 -5443.064,E2 -5443.064} C_VEL
LIN {X 0,Y 509.908,Z 485.723,A -85,B 0,C 180,E1 -5444.531,E2 -5444.531} C_VEL
LIN {X 0,Y 510.962,Z 491.92,A -85,B 0,C 180,E1 -5447.626,E2 -5447.626} C_VEL
LIN {X 0,Y 511.065,Z 496.592,A -85,B 0,C 180,E1 -5449.735,E2 -5449.735} C_VEL
LIN {X 0,Y 510.777,Z 503.839,A -85,B 0,C 180,E1 -5452.742,E2 -5452.742} C_VEL
LIN {X 0,Y 510.548,Z 511.373,A -85,B 0,C 180,E1 -5455.683,E2 -5455.683} C_VEL
LIN {X 0,Y 510.336,Z 520.353,A -85,B 0,C 180,E1 -5458.995,E2 -5458.995} C_VEL
LIN {X 0,Y 510.134,Z 529.12,A -85,B 0,C 180,E1 -5462.069,E2 -5462.069} C_VEL
LIN {X 0,Y 509.98,Z 536.811,A -85,B 0,C 180,E1 -5464.71,E2 -5464.71} C_VEL
LIN {X 0,Y 509.83,Z 546.34,A -85,B 0,C 180,E1 -5467.804,E2 -5467.804} C_VEL
LIN {X 0,Y 509.731,Z 553.417,A -85,B 0,C 180,E1 -5470.089,E2 -5470.089} C_VEL
LIN {X 0,Y 513.96,Z 571.801,A -85,B 0,C 180,E1 -5470.616,E2 -5470.616} C_VEL
LIN {X 0,Y 513.556,Z 587.282,A -85,B 0,C 180,E1 -5471.079,E2 -5471.079} C_VEL
LIN {X 0,Y 513.09,Z 602.081,A -85,B 0,C 180,E1 -5471.688,E2 -5471.688} C_VEL
LIN {X 0,Y 512.615,Z 616.313,A -85,B 0,C 180,E1 -5472.445,E2 -5472.445} C_VEL
LIN {X 0,Y 512.03,Z 630.041,A -85,B 0,C 180,E1 -5473.35,E2 -5473.35} C_VEL
LIN {X 0,Y 511.501,Z 642.796,A -85,B 0,C 180,E1 -5474.374,E2 -5474.374} C_VEL
LIN {X 0,Y 510.962,Z 654.164,A -85,B 0,C 180,E1 -5475.462,E2 -5475.462} C_VEL
LIN {X 0,Y 510.504,Z 664.763,A -85,B 0,C 180,E1 -5476.668,E2 -5476.668} C_VEL
LIN {X 0,Y 510.002,Z 675.013,A -85,B 0,C 180,E1 -5478.07,E2 -5478.07} C_VEL
LIN {X 0,Y 509.818,Z 683.53,A -85,B 0,C 180,E1 -5479.475,E2 -5479.475} C_VEL
LIN {X 0,Y 509.537,Z 690.614,A -85,B 0,C 180,E1 -5480.873,E2 -5480.873} C_VEL
LIN {X 0,Y 509.352,Z 697.182,A -85,B 0,C 180,E1 -5482.468,E2 -5482.468} C_VEL
LIN {X 0,Y 509.294,Z 702.319,A -85,B 0,C 180,E1 -5484.059,E2 -5484.059} C_VEL
LIN {X 0,Y 509.159,Z 705.29,A -85,B 0,C 180,E1 -5485.249,E2 -5485.249} C_VEL
LIN {X 0,Y 509.188,Z 708.183,A -85,B 0,C 180,E1 -5486.835,E2 -5486.835} C_VEL
LIN {X 0,Y 509.109,Z 709.909,A -85,B 0,C 180,E1 -5488.418,E2 -5488.418} C_VEL
LIN {X 0,Y 509.062,Z 710.5,A -85,B 0,C 180,E1 -5490,E2 -5490} C_VEL
LIN {X 0,Y 509.109,Z 709.907,A -85,B 0,C 180,E1 -5491.582,E2 -5491.582} C_VEL
LIN {X 0,Y 509.188,Z 708.18,A -85,B 0,C 180,E1 -5493.164,E2 -5493.164} C_VEL
LIN {X 0,Y 509.158,Z 705.289,A -85,B 0,C 180,E1 -5494.75,E2 -5494.75} C_VEL
LIN {X 0,Y 509.26,Z 701.167,A -85,B 0,C 180,E1 -5496.338,E2 -5496.338} C_VEL
LIN {X 0,Y 509.411,Z 695.703,A -85,B 0,C 180,E1 -5497.929,E2 -5497.929} C_VEL
LIN {X 0,Y 509.56,Z 688.746,A -85,B 0,C 180,E1 -5499.526,E2 -5499.526} C_VEL
LIN {X 0,Y 509.954,Z 680.084,A -85,B 0,C 180,E1 -5501.124,E2 -5501.124} C_VEL
LIN {X 0,Y 510.237,Z 671.026,A -85,B 0,C 180,E1 -5502.509,E2 -5502.509} C_VEL
LIN {X 0,Y 510.656,Z 661.5,A -85,B 0,C 180,E1 -5503.733,E2 -5503.733} C_VEL
LIN {X 0,Y 511.165,Z 649.208,A -85,B 0,C 180,E1 -5505.04,E2 -5505.04} C_VEL
LIN {X 0,Y 511.734,Z 636.679,A -85,B 0,C 180,E1 -5506.147,E2 -5506.147} C_VEL
LIN {X 0,Y 512.334,Z 622.831,A -85,B 0,C 180,E1 -5507.152,E2 -5507.152} C_VEL
LIN {X 0,Y 512.838,Z 609.242,A -85,B 0,C 180,E1 -5507.959,E2 -5507.959} C_VEL
LIN {X 0,Y 513.426,Z 594.727,A -85,B 0,C 180,E1 -5508.638,E2 -5508.638} C_VEL
LIN {X 0,Y 513.8,Z 579.228,A -85,B 0,C 180,E1 -5509.187,E2 -5509.187} C_VEL
LIN {X 0,Y 513.887,Z 571.597,A -85,B 0,C 180,E1 -5509.396,E2 -5509.396} C_VEL
LIN {X 0,Y 509.831,Z 554.538,A -85,B 0,C 180,E1 -5509.884,E2 -5509.884} C_VEL
LIN {X 0,Y 509.733,Z 553.637,A -85,B 0,C 180,E1 -5509.931,E2 -5509.931} C_VEL
LIN {X 0,Y 509.938,Z 543.948,A -85,B 0,C 180,E1 -5513.127,E2 -5513.127} C_VEL
LIN {X 0,Y 510.107,Z 534.071,A -85,B 0,C 180,E1 -5516.423,E2 -5516.423} C_VEL
LIN {X 0,Y 510.294,Z 525.939,A -85,B 0,C 180,E1 -5519.269,E2 -5519.269} C_VEL
LIN {X 0,Y 510.45,Z 518.416,A -85,B 0,C 180,E1 -5522.01,E2 -5522.01} C_VEL
LIN {X 0,Y 510.68,Z 510.909,A -85,B 0,C 180,E1 -5524.827,E2 -5524.827} C_VEL
LIN {X 0,Y 510.969,Z 503.468,A -85,B 0,C 180,E1 -5527.738,E2 -5527.738} C_VEL
LIN {X 0,Y 511.235,Z 497.331,A -85,B 0,C 180,E1 -5530.248,E2 -5530.248} C_VEL
LIN {X 0,Y 511.16,Z 493.135,A -85,B 0,C 180,E1 -5532.059,E2 -5532.059} C_VEL
LIN {X 0,Y 510.214,Z 487.603,A -85,B 0,C 180,E1 -5534.627,E2 -5534.627} C_VEL
LIN {X 0,Y 509.874,Z 485.601,A -85,B 0,C 180,E1 -5535.595,E2 -5535.595} C_VEL
LIN {X 0,Y 509.865,Z 485.602,A -85,B 0,C 180,E1 -5538.576,E2 -5538.576} C_VEL
LIN {X 0,Y 509.848,Z 485.604,A -85,B 0,C 180,E1 -5541.785,E2 -5541.785} C_VEL
LIN {X 0,Y 509.838,Z 485.603,A -85,B 0,C 180,E1 -5544.623,E2 -5544.623} C_VEL
LIN {X 0,Y 509.857,Z 485.604,A -85,B 0,C 180,E1 -5547.481,E2 -5547.481} C_VEL
LIN {X 0,Y 509.872,Z 485.598,A -85,B 0,C 180,E1 -5550.268,E2 -5550.268} C_VEL
LIN {X 0,Y 509.878,Z 485.599,A -85,B 0,C 180,E1 -5552.944,E2 -5552.944} C_VEL
LIN {X 0,Y 509.86,Z 485.602,A -85,B 0,C 180,E1 -5555.574,E2 -5555.574} C_VEL
LIN {X 0,Y 509.812,Z 485.607,A -85,B 0,C 180,E1 -5558.148,E2 -5558.148} C_VEL
LIN {X 0,Y 509.856,Z 485.601,A -85,B 0,C 180,E1 -5560.682,E2 -5560.682} C_VEL
LIN {X 0,Y 509.877,Z 485.601,A -85,B 0,C 180,E1 -5563.175,E2 -5563.175} C_VEL
LIN {X 0,Y 509.854,Z 485.602,A -85,B 0,C 180,E1 -5565.634,E2 -5565.634} C_VEL
LIN {X 0,Y 509.915,Z 485.594,A -85,B 0,C 180,E1 -5568.875,E2 -5568.875} C_VEL
LIN {X 0,Y 509.942,Z 485.59,A -85,B 0,C 180,E1 -5572.079,E2 -5572.079} C_VEL
LIN {X 0,Y 509.985,Z 485.583,A -85,B 0,C 180,E1 -5574.465,E2 -5574.465} C_VEL
LIN {X 0,Y 510.047,Z 485.579,A -85,B 0,C 180,E1 -5577.631,E2 -5577.631} C_VEL
LIN {X 0,Y 510.056,Z 485.577,A -85,B 0,C 180,E1 -5580.79,E2 -5580.79} C_VEL
LIN {X 0,Y 509.953,Z 485.59,A -85,B 0,C 180,E1 -5583.16,E2 -5583.16} C_VEL
LIN {X 0,Y 509.974,Z 485.586,A -85,B 0,C 180,E1 -5586.33,E2 -5586.33} C_VEL
LIN {X 0,Y 509.91,Z 485.594,A -85,B 0,C 180,E1 -5588.721,E2 -5588.721} C_VEL
LIN {X 0,Y 509.895,Z 485.597,A -85,B 0,C 180,E1 -5591.932,E2 -5591.932} C_VEL
LIN {X 0,Y 509.884,Z 485.599,A -85,B 0,C 180,E1 -5595.242,E2 -5595.242} C_VEL
LIN {X 0,Y 509.88,Z 485.6,A -85,B 0,C 180,E1 -5598.002,E2 -5598.002} C_VEL
LIN {X 0,Y 509.842,Z 485.603,A -85,B 0,C 180,E1 -5601.002,E2 -5601.002} C_VEL
LIN {X 0,Y 509.828,Z 485.607,A -85,B 0,C 180,E1 -5603.564,E2 -5603.564} C_VEL
LIN {X 0,Y 509.907,Z 485.594,A -85,B 0,C 180,E1 -5606.38,E2 -5606.38} C_VEL
LIN {X 0,Y 509.879,Z 485.597,A -85,B 0,C 180,E1 -5608.845,E2 -5608.845} C_VEL
LIN {X 0,Y 509.82,Z 485.608,A -85,B 0,C 180,E1 -5611.591,E2 -5611.591} C_VEL
LIN {X 0,Y 509.849,Z 485.603,A -85,B 0,C 180,E1 -5614.414,E2 -5614.414} C_VEL
LIN {X 0,Y 509.814,Z 485.607,A -85,B 0,C 180,E1 -5617.342,E2 -5617.342} C_VEL
LIN {X 0,Y 509.875,Z 485.599,A -85,B 0,C 180,E1 -5620.379,E2 -5620.379} C_VEL
LIN {X 0,Y 509.837,Z 485.604,A -85,B 0,C 180,E1 -5623.065,E2 -5623.065} C_VEL
LIN {X 0,Y 509.828,Z 485.607,A -85,B 0,C 180,E1 -5625.793,E2 -5625.793} C_VEL
LIN {X 0,Y 509.864,Z 485.599,A -85,B 0,C 180,E1 -5628.577,E2 -5628.577} C_VEL
LIN {X 0,Y 509.858,Z 485.602,A -85,B 0,C 180,E1 -5631.664,E2 -5631.664} C_VEL
LIN {X 0,Y 509.829,Z 485.605,A -85,B 0,C 180,E1 -5633.75,E2 -5633.75} C_VEL
LIN {X 0,Y 509.164,Z 485.688,A -85,B 0,C 180,E1 -5634.409,E2 -5634.409} C_VEL
LIN {X 0,Y 506.346,Z 486.04,A -85,B 0,C 180,E1 -5635.481,E2 -5635.481} C_VEL
LIN {X 0,Y 503.953,Z 486.339,A -85,B 0,C 180,E1 -5636.345,E2 -5636.345} C_VEL
LIN {X 0,Y 502.905,Z 486.469,A -85,B 0,C 180,E1 -5637.011,E2 -5637.011} C_VEL
LIN {X 0,Y 502.808,Z 486.479,A -85,B 0,C 180,E1 -5637.237,E2 -5637.237} C_VEL
LIN {X 0,Y 502.816,Z 486.479,A -85,B 0,C 180,E1 -5640.066,E2 -5640.066} C_VEL
LIN {X 0,Y 502.837,Z 486.475,A -85,B 0,C 180,E1 -5642.534,E2 -5642.534} C_VEL
LIN {X 0,Y 502.832,Z 486.477,A -85,B 0,C 180,E1 -5645.299,E2 -5645.299} C_VEL
LIN {X 0,Y 502.788,Z 486.483,A -85,B 0,C 180,E1 -5647.828,E2 -5647.828} C_VEL
LIN {X 0,Y 502.828,Z 486.475,A -85,B 0,C 180,E1 -5650.401,E2 -5650.401} C_VEL
LIN {X 0,Y 502.838,Z 486.474,A -85,B 0,C 180,E1 -5652.933,E2 -5652.933} C_VEL
LIN {X 0,Y 502.849,Z 486.476,A -85,B 0,C 180,E1 -5655.43,E2 -5655.43} C_VEL
LIN {X 0,Y 502.882,Z 486.47,A -85,B 0,C 180,E1 -5658.718,E2 -5658.718} C_VEL
LIN {X 0,Y 502.885,Z 486.472,A -85,B 0,C 180,E1 -5661.967,E2 -5661.967} C_VEL
LIN {X 0,Y 502.943,Z 486.462,A -85,B 0,C 180,E1 -5664.387,E2 -5664.387} C_VEL
LIN {X 0,Y 503.031,Z 486.454,A -85,B 0,C 180,E1 -5667.598,E2 -5667.598} C_VEL
LIN {X 0,Y 503.034,Z 486.452,A -85,B 0,C 180,E1 -5670,E2 -5670} C_VEL
LIN {X 0,Y 502.886,Z 486.471,A -85,B 0,C 180,E1 -5672.403,E2 -5672.403} C_VEL
LIN {X 0,Y 502.658,Z 486.501,A -85,B 0,C 180,E1 -5674.813,E2 -5674.813} C_VEL
LIN {X 0,Y 502.463,Z 486.704,A -85,B 0,C 180,E1 -5675.619,E2 -5675.619} C_VEL
LIN {X 0,Y 502.435,Z 488.917,A -85,B 0,C 180,E1 -5678.041,E2 -5678.041} C_VEL
LIN {X 0,Y 502.389,Z 492.276,A -85,B 0,C 180,E1 -5681.693,E2 -5681.693} C_VEL
LIN {X 0,Y 502.308,Z 495.456,A -85,B 0,C 180,E1 -5685.112,E2 -5685.112} C_VEL
LIN {X 0,Y 502.211,Z 498.064,A -85,B 0,C 180,E1 -5687.931,E2 -5687.931} C_VEL
LIN {X 0,Y 502.198,Z 499.906,A -85,B 0,C 180,E1 -5689.882,E2 -5689.882} C_VEL
LIN {X 0,Y 506.3,Z 514.428,A -85,B 0,C 180,E1 -5690.372,E2 -5690.372} C_VEL
LIN {X 0,Y 507.237,Z 519.51,A -85,B 0,C 180,E1 -5690.558,E2 -5690.558} C_VEL
LIN {X 0,Y 506.787,Z 534.75,A -85,B 0,C 180,E1 -5691.088,E2 -5691.088} C_VEL
LIN {X 0,Y 506.313,Z 548.689,A -85,B 0,C 180,E1 -5691.738,E2 -5691.738} C_VEL
LIN {X 0,Y 505.753,Z 561.21,A -85,B 0,C 180,E1 -5692.466,E2 -5692.466} C_VEL
LIN {X 0,Y 505.123,Z 574.632,A -85,B 0,C 180,E1 -5693.424,E2 -5693.424} C_VEL
LIN {X 0,Y 504.517,Z 586.858,A -85,B 0,C 180,E1 -5694.483,E2 -5694.483} C_VEL
LIN {X 0,Y 503.943,Z 597.819,A -85,B 0,C 180,E1 -5695.615,E2 -5695.615} C_VEL
LIN {X 0,Y 503.464,Z 607.698,A -85,B 0,C 180,E1 -5696.821,E2 -5696.821} C_VEL
LIN {X 0,Y 503.053,Z 616.561,A -85,B 0,C 180,E1 -5698.105,E2 -5698.105} C_VEL
LIN {X 0,Y 502.678,Z 625.182,A -85,B 0,C 180,E1 -5699.598,E2 -5699.598} C_VEL
LIN {X 0,Y 502.414,Z 632.614,A -85,B 0,C 180,E1 -5701.169,E2 -5701.169} C_VEL
LIN {X 0,Y 502.224,Z 637.768,A -85,B 0,C 180,E1 -5702.507,E2 -5702.507} C_VEL
LIN {X 0,Y 502.121,Z 642.541,A -85,B 0,C 180,E1 -5704.046,E2 -5704.046} C_VEL
LIN {X 0,Y 501.995,Z 646.378,A -85,B 0,C 180,E1 -5705.707,E2 -5705.707} C_VEL
LIN {X 0,Y 501.928,Z 648.52,A -85,B 0,C 180,E1 -5707.049,E2 -5707.049} C_VEL
LIN {X 0,Y 501.948,Z 649.875,A -85,B 0,C 180,E1 -5708.363,E2 -5708.363} C_VEL
LIN {X 0,Y 501.95,Z 650.499,A -85,B 0,C 180,E1 -5710.095,E2 -5710.095} C_VEL
LIN {X 0,Y 501.941,Z 650.213,A -85,B 0,C 180,E1 -5711.153,E2 -5711.153} C_VEL
LIN {X 0,Y 501.972,Z 649.438,A -85,B 0,C 180,E1 -5712.224,E2 -5712.224} C_VEL
LIN {X 0,Y 501.997,Z 648.15,A -85,B 0,C 180,E1 -5713.314,E2 -5713.314} C_VEL
LIN {X 0,Y 502.089,Z 645.135,A -85,B 0,C 180,E1 -5714.98,E2 -5714.98} C_VEL
LIN {X 0,Y 502.181,Z 640.643,A -85,B 0,C 180,E1 -5716.705,E2 -5716.705} C_VEL
LIN {X 0,Y 502.313,Z 634.845,A -85,B 0,C 180,E1 -5718.378,E2 -5718.378} C_VEL
LIN {X 0,Y 502.57,Z 627.885,A -85,B 0,C 180,E1 -5719.963,E2 -5719.963} C_VEL
LIN {X 0,Y 502.903,Z 619.595,A -85,B 0,C 180,E1 -5721.498,E2 -5721.498} C_VEL
LIN {X 0,Y 503.379,Z 610.262,A -85,B 0,C 180,E1 -5722.923,E2 -5722.923} C_VEL
LIN {X 0,Y 503.885,Z 599.748,A -85,B 0,C 180,E1 -5724.263,E2 -5724.263} C_VEL
LIN {X 0,Y 504.476,Z 588.333,A -85,B 0,C 180,E1 -5725.476,E2 -5725.476} C_VEL
LIN {X 0,Y 505.088,Z 575.595,A -85,B 0,C 180,E1 -5726.601,E2 -5726.601} C_VEL
LIN {X 0,Y 505.726,Z 561.907,A -85,B 0,C 180,E1 -5727.59,E2 -5727.59} C_VEL
LIN {X 0,Y 506.308,Z 548.003,A -85,B 0,C 180,E1 -5728.398,E2 -5728.398} C_VEL
LIN {X 0,Y 506.876,Z 533.005,A -85,B 0,C 180,E1 -5729.077,E2 -5729.077} C_VEL
LIN {X 0,Y 507.217,Z 518.319,A -85,B 0,C 180,E1 -5729.573,E2 -5729.573} C_VEL
LIN {X 0,Y 503.78,Z 505.184,A -85,B 0,C 180,E1 -5730.038,E2 -5730.038} C_VEL
LIN {X 0,Y 502.211,Z 500.279,A -85,B 0,C 180,E1 -5730.212,E2 -5730.212} C_VEL
LIN {X 0,Y 502.265,Z 497.35,A -85,B 0,C 180,E1 -5733.575,E2 -5733.575} C_VEL
LIN {X 0,Y 502.297,Z 495.184,A -85,B 0,C 180,E1 -5736.061,E2 -5736.061} C_VEL
LIN {X 0,Y 502.377,Z 492.915,A -85,B 0,C 180,E1 -5738.67,E2 -5738.67} C_VEL
LIN {X 0,Y 502.533,Z 489.957,A -85,B 0,C 180,E1 -5742.081,E2 -5742.081} C_VEL
LIN {X 0,Y 502.571,Z 487.083,A -85,B 0,C 180,E1 -5745.421,E2 -5745.421} C_VEL
LIN {X 0,Y 502.571,Z 486.513,A -85,B 0,C 180,E1 -5746.247,E2 -5746.247} C_VEL
LIN {X 0,Y 502.851,Z 486.474,A -85,B 0,C 180,E1 -5748.716,E2 -5748.716} C_VEL
LIN {X 0,Y 502.899,Z 486.47,A -85,B 0,C 180,E1 -5751.966,E2 -5751.966} C_VEL
LIN {X 0,Y 502.939,Z 486.462,A -85,B 0,C 180,E1 -5754.386,E2 -5754.386} C_VEL
LIN {X 0,Y 503.022,Z 486.454,A -85,B 0,C 180,E1 -5757.597,E2 -5757.597} C_VEL
LIN {X 0,Y 503.023,Z 486.452,A -85,B 0,C 180,E1 -5760,E2 -5760} C_VEL
LIN {X 0,Y 503.02,Z 486.449,A -85,B 0,C 180,E1 -5762.402,E2 -5762.402} C_VEL
LIN {X 0,Y 502.944,Z 486.462,A -85,B 0,C 180,E1 -5765.613,E2 -5765.613} C_VEL
LIN {X 0,Y 502.898,Z 486.464,A -85,B 0,C 180,E1 -5768.033,E2 -5768.033} C_VEL
LIN {X 0,Y 502.877,Z 486.47,A -85,B 0,C 180,E1 -5771.283,E2 -5771.283} C_VEL
LIN {X 0,Y 502.84,Z 486.475,A -85,B 0,C 180,E1 -5774.571,E2 -5774.571} C_VEL
LIN {X 0,Y 502.857,Z 486.469,A -85,B 0,C 180,E1 -5777.907,E2 -5777.907} C_VEL
LIN {X 0,Y 502.825,Z 486.479,A -85,B 0,C 180,E1 -5780.536,E2 -5780.536} C_VEL
LIN {X 0,Y 502.793,Z 486.477,A -85,B 0,C 180,E1 -5783.04,E2 -5783.04} C_VEL
LIN {X 0,Y 502.838,Z 486.473,A -85,B 0,C 180,E1 -5785.675,E2 -5785.675} C_VEL
LIN {X 0,Y 502.839,Z 486.476,A -85,B 0,C 180,E1 -5788.372,E2 -5788.372} C_VEL
LIN {X 0,Y 502.794,Z 486.481,A -85,B 0,C 180,E1 -5791.5,E2 -5791.5} C_VEL
LIN {X 0,Y 502.803,Z 486.477,A -85,B 0,C 180,E1 -5794.445,E2 -5794.445} C_VEL
LIN {X 0,Y 502.778,Z 486.483,A -85,B 0,C 180,E1 -5797.178,E2 -5797.178} C_VEL
LIN {X 0,Y 502.786,Z 486.48,A -85,B 0,C 180,E1 -5800.015,E2 -5800.015} C_VEL
LIN {X 0,Y 502.8,Z 486.48,A -85,B 0,C 180,E1 -5802.199,E2 -5802.199} C_VEL
LIN {X 0,Y 502.846,Z 486.636,A -85,B 0,C 180,E1 -5804.203,E2 -5804.203} C_VEL
LIN {X 0,Y 503.767,Z 491.797,A -85,B 0,C 180,E1 -5806.875,E2 -5806.875} C_VEL
LIN {X 0,Y 504.174,Z 495.948,A -85,B 0,C 180,E1 -5808.828,E2 -5808.828} C_VEL
LIN {X 0,Y 503.934,Z 501.741,A -85,B 0,C 180,E1 -5811.351,E2 -5811.351} C_VEL
LIN {X 0,Y 503.648,Z 509.735,A -85,B 0,C 180,E1 -5814.613,E2 -5814.613} C_VEL
LIN {X 0,Y 503.4,Z 515.986,A -85,B 0,C 180,E1 -5817.011,E2 -5817.011} C_VEL
LIN {X 0,Y 503.249,Z 522.305,A -85,B 0,C 180,E1 -5819.354,E2 -5819.354} C_VEL
LIN {X 0,Y 503.071,Z 530.039,A -85,B 0,C 180,E1 -5822.1,E2 -5822.1} C_VEL
LIN {X 0,Y 502.921,Z 537.736,A -85,B 0,C 180,E1 -5824.772,E2 -5824.772} C_VEL
LIN {X 0,Y 502.761,Z 546.943,A -85,B 0,C 180,E1 -5827.826,E2 -5827.826} C_VEL
LIN {X 0,Y 502.68,Z 553.133,A -85,B 0,C 180,E1 -5829.813,E2 -5829.813} C_VEL
LIN {X 0,Y 505.759,Z 566.665,A -85,B 0,C 180,E1 -5830.185,E2 -5830.185} C_VEL
LIN {X 0,Y 507.204,Z 574.178,A -85,B 0,C 180,E1 -5830.43,E2 -5830.43} C_VEL
LIN {X 0,Y 506.75,Z 588.247,A -85,B 0,C 180,E1 -5830.875,E2 -5830.875} C_VEL
LIN {X 0,Y 506.26,Z 602.573,A -85,B 0,C 180,E1 -5831.485,E2 -5831.485} C_VEL
LIN {X 0,Y 505.68,Z 617.419,A -85,B 0,C 180,E1 -5832.301,E2 -5832.301} C_VEL
LIN {X 0,Y 505.071,Z 630.865,A -85,B 0,C 180,E1 -5833.218,E2 -5833.218} C_VEL
LIN {X 0,Y 504.471,Z 644.209,A -85,B 0,C 180,E1 -5834.329,E2 -5834.329} C_VEL
LIN {X 0,Y 503.889,Z 655.592,A -85,B 0,C 180,E1 -5835.46,E2 -5835.46} C_VEL
LIN {X 0,Y 503.421,Z 665.959,A -85,B 0,C 180,E1 -5836.682,E2 -5836.682} C_VEL
LIN {X 0,Y 502.947,Z 676.447,A -85,B 0,C 180,E1 -5838.158,E2 -5838.158} C_VEL
LIN {X 0,Y 502.708,Z 684.532,A -85,B 0,C 180,E1 -5839.528,E2 -5839.528} C_VEL
LIN {X 0,Y 502.467,Z 690.598,A -85,B 0,C 180,E1 -5840.744,E2 -5840.744} C_VEL
LIN {X 0,Y 502.301,Z 697.182,A -85,B 0,C 180,E1 -5842.361,E2 -5842.361} C_VEL
LIN {X 0,Y 502.178,Z 701.793,A -85,B 0,C 180,E1 -5843.779,E2 -5843.779} C_VEL
LIN {X 0,Y 502.081,Z 705.289,A -85,B 0,C 180,E1 -5845.182,E2 -5845.182} C_VEL
LIN {X 0,Y 502.107,Z 708.183,A -85,B 0,C 180,E1 -5846.79,E2 -5846.79} C_VEL
LIN {X 0,Y 502.033,Z 709.908,A -85,B 0,C 180,E1 -5848.395,E2 -5848.395} C_VEL
LIN {X 0,Y 501.977,Z 710.5,A -85,B 0,C 180,E1 -5850,E2 -5850} C_VEL
LIN {X 0,Y 502.032,Z 709.906,A -85,B 0,C 180,E1 -5851.604,E2 -5851.604} C_VEL
LIN {X 0,Y 502.107,Z 708.179,A -85,B 0,C 180,E1 -5853.209,E2 -5853.209} C_VEL
LIN {X 0,Y 502.081,Z 705.289,A -85,B 0,C 180,E1 -5854.817,E2 -5854.817} C_VEL
LIN {X 0,Y 502.184,Z 701.042,A -85,B 0,C 180,E1 -5856.468,E2 -5856.468} C_VEL
LIN {X 0,Y 502.339,Z 695.702,A -85,B 0,C 180,E1 -5858.042,E2 -5858.042} C_VEL
LIN {X 0,Y 502.466,Z 690.597,A -85,B 0,C 180,E1 -5859.256,E2 -5859.256} C_VEL
LIN {X 0,Y 502.759,Z 683.406,A -85,B 0,C 180,E1 -5860.673,E2 -5860.673} C_VEL
LIN {X 0,Y 503.038,Z 674.76,A -85,B 0,C 180,E1 -5862.096,E2 -5862.096} C_VEL
LIN {X 0,Y 503.508,Z 664.366,A -85,B 0,C 180,E1 -5863.52,E2 -5863.52} C_VEL
LIN {X 0,Y 503.97,Z 653.741,A -85,B 0,C 180,E1 -5864.743,E2 -5864.743} C_VEL
LIN {X 0,Y 504.554,Z 641.635,A -85,B 0,C 180,E1 -5865.913,E2 -5865.913} C_VEL
LIN {X 0,Y 505.151,Z 629.668,A -85,B 0,C 180,E1 -5866.883,E2 -5866.883} C_VEL
LIN {X 0,Y 505.792,Z 615.954,A -85,B 0,C 180,E1 -5867.799,E2 -5867.799} C_VEL
LIN {X 0,Y 506.335,Z 601.762,A -85,B 0,C 180,E1 -5868.564,E2 -5868.564} C_VEL
LIN {X 0,Y 506.881,Z 586.353,A -85,B 0,C 180,E1 -5869.202,E2 -5869.202} C_VEL
LIN {X 0,Y 507.061,Z 572.362,A -85,B 0,C 180,E1 -5869.636,E2 -5869.636} C_VEL
LIN {X 0,Y 503.102,Z 555.623,A -85,B 0,C 180,E1 -5870.138,E2 -5870.138} C_VEL
LIN {X 0,Y 502.69,Z 553.324,A -85,B 0,C 180,E1 -5870.191,E2 -5870.191} C_VEL
LIN {X 0,Y 502.881,Z 543.65,A -85,B 0,C 180,E1 -5873.471,E2 -5873.471} C_VEL
LIN {X 0,Y 503.052,Z 534.402,A -85,B 0,C 180,E1 -5876.604,E2 -5876.604} C_VEL
LIN {X 0,Y 503.302,Z 525.878,A -85,B 0,C 180,E1 -5879.646,E2 -5879.646} C_VEL
LIN {X 0,Y 503.499,Z 518.167,A -85,B 0,C 180,E1 -5882.505,E2 -5882.505} C_VEL
LIN {X 0,Y 503.722,Z 510.679,A -85,B 0,C 180,E1 -5885.38,E2 -5885.38} C_VEL
LIN {X 0,Y 504.086,Z 502.479,A -85,B 0,C 180,E1 -5888.67,E2 -5888.67} C_VEL
LIN {X 0,Y 504.325,Z 496.521,A -85,B 0,C 180,E1 -5891.192,E2 -5891.192} C_VEL
LIN {X 0,Y 503.874,Z 492.277,A -85,B 0,C 180,E1 -5893.112,E2 -5893.112} C_VEL
LIN {X 0,Y 502.793,Z 486.483,A -85,B 0,C 180,E1 -5895.921,E2 -5895.921} C_VEL
LIN {X 0,Y 502.824,Z 486.479,A -85,B 0,C 180,E1 -5899.003,E2 -5899.003} C_VEL
LIN {X 0,Y 502.789,Z 486.484,A -85,B 0,C 180,E1 -5902.046,E2 -5902.046} C_VEL
LIN {X 0,Y 502.802,Z 486.48,A -85,B 0,C 180,E1 -5905.035,E2 -5905.035} C_VEL
LIN {X 0,Y 502.779,Z 486.483,A -85,B 0,C 180,E1 -5907.915,E2 -5907.915} C_VEL
LIN {X 0,Y 502.83,Z 486.476,A -85,B 0,C 180,E1 -5910.713,E2 -5910.713} C_VEL
LIN {X 0,Y 502.871,Z 486.473,A -85,B 0,C 180,E1 -5913.435,E2 -5913.435} C_VEL
LIN {X 0,Y 502.782,Z 486.484,A -85,B 0,C 180,E1 -5916.086,E2 -5916.086} C_VEL
LIN {X 0,Y 502.774,Z 486.484,A -85,B 0,C 180,E1 -5918.689,E2 -5918.689} C_VEL
LIN {X 0,Y 502.821,Z 486.478,A -85,B 0,C 180,E1 -5921.248,E2 -5921.248} C_VEL
LIN {X 0,Y 502.814,Z 486.48,A -85,B 0,C 180,E1 -5923.767,E2 -5923.767} C_VEL
LIN {X 0,Y 502.821,Z 486.478,A -85,B 0,C 180,E1 -5926.255,E2 -5926.255} C_VEL
LIN {X 0,Y 502.884,Z 486.47,A -85,B 0,C 180,E1 -5928.717,E2 -5928.717} C_VEL
LIN {X 0,Y 502.892,Z 486.469,A -85,B 0,C 180,E1 -5931.967,E2 -5931.967} C_VEL
LIN {X 0,Y 502.939,Z 486.461,A -85,B 0,C 180,E1 -5934.387,E2 -5934.387} C_VEL
LIN {X 0,Y 503.017,Z 486.454,A -85,B 0,C 180,E1 -5937.598,E2 -5937.598} C_VEL
LIN {X 0,Y 503.016,Z 486.454,A -85,B 0,C 180,E1 -5940,E2 -5940} C_VEL
LIN {X 0,Y 503.017,Z 486.453,A -85,B 0,C 180,E1 -5942.403,E2 -5942.403} C_VEL
LIN {X 0,Y 502.955,Z 486.462,A -85,B 0,C 180,E1 -5945.614,E2 -5945.614} C_VEL
LIN {X 0,Y 502.893,Z 486.47,A -85,B 0,C 180,E1 -5948.034,E2 -5948.034} C_VEL
LIN {X 0,Y 502.872,Z 486.472,A -85,B 0,C 180,E1 -5951.284,E2 -5951.284} C_VEL
LIN {X 0,Y 502.836,Z 486.475,A -85,B 0,C 180,E1 -5954.571,E2 -5954.571} C_VEL
LIN {X 0,Y 502.853,Z 486.475,A -85,B 0,C 180,E1 -5957.908,E2 -5957.908} C_VEL
LIN {X 0,Y 502.82,Z 486.478,A -85,B 0,C 180,E1 -5960.537,E2 -5960.537} C_VEL
LIN {X 0,Y 502.788,Z 486.482,A -85,B 0,C 180,E1 -5963.041,E2 -5963.041} C_VEL
LIN {X 0,Y 502.834,Z 486.478,A -85,B 0,C 180,E1 -5965.676,E2 -5965.676} C_VEL
LIN {X 0,Y 502.836,Z 486.475,A -85,B 0,C 180,E1 -5968.373,E2 -5968.373} C_VEL
LIN {X 0,Y 502.791,Z 486.484,A -85,B 0,C 180,E1 -5971.501,E2 -5971.501} C_VEL
LIN {X 0,Y 502.802,Z 486.48,A -85,B 0,C 180,E1 -5974.446,E2 -5974.446} C_VEL
LIN {X 0,Y 502.776,Z 486.485,A -85,B 0,C 180,E1 -5977.18,E2 -5977.18} C_VEL
LIN {X 0,Y 502.831,Z 486.478,A -85,B 0,C 180,E1 -5980.012,E2 -5980.012} C_VEL
LIN {X 0,Y 502.823,Z 486.479,A -85,B 0,C 180,E1 -5982.203,E2 -5982.203} C_VEL
LIN {X 0,Y 502.797,Z 486.482,A -85,B 0,C 180,E1 -5985.469,E2 -5985.469} C_VEL
LIN {X 0,Y 502.833,Z 486.478,A -85,B 0,C 180,E1 -5987.866,E2 -5987.866} C_VEL
LIN {X 0,Y 502.82,Z 486.477,A -85,B 0,C 180,E1 -5991.027,E2 -5991.027} C_VEL
LIN {X 0,Y 502.783,Z 486.483,A -85,B 0,C 180,E1 -5994.169,E2 -5994.169} C_VEL
LIN {X 0,Y 502.808,Z 486.479,A -85,B 0,C 180,E1 -5997.237,E2 -5997.237} C_VEL
LIN {X 0,Y 502.108,Z 486.568,A -85,B 0,C 180,E1 -5997.905,E2 -5997.905} C_VEL
LIN {X 0,Y 499.243,Z 486.924,A -85,B 0,C 180,E1 -5998.991,E2 -5998.991} C_VEL
LIN {X 0,Y 496.848,Z 487.224,A -85,B 0,C 180,E1 -5999.866,E2 -5999.866} C_VEL
LIN {X 0,Y 495.832,Z 487.346,A -85,B 0,C 180,E1 -6000.542,E2 -6000.542} C_VEL
LIN {X 0,Y 495.755,Z 487.356,A -85,B 0,C 180,E1 -6000.77,E2 -6000.77} C_VEL
LIN {X 0,Y 495.802,Z 487.353,A -85,B 0,C 180,E1 -6003.934,E2 -6003.934} C_VEL
LIN {X 0,Y 495.768,Z 487.357,A -85,B 0,C 180,E1 -6007.139,E2 -6007.139} C_VEL
LIN {X 0,Y 495.775,Z 487.355,A -85,B 0,C 180,E1 -6010.111,E2 -6010.111} C_VEL
LIN {X 0,Y 495.791,Z 487.352,A -85,B 0,C 180,E1 -6012.682,E2 -6012.682} C_VEL
LIN {X 0,Y 495.794,Z 487.353,A -85,B 0,C 180,E1 -6015.218,E2 -6015.218} C_VEL
LIN {X 0,Y 495.856,Z 487.345,A -85,B 0,C 180,E1 -6018.556,E2 -6018.556} C_VEL
LIN {X 0,Y 495.841,Z 487.349,A -85,B 0,C 180,E1 -6021.852,E2 -6021.852} C_VEL
LIN {X 0,Y 495.901,Z 487.34,A -85,B 0,C 180,E1 -6024.307,E2 -6024.307} C_VEL
LIN {X 0,Y 495.999,Z 487.33,A -85,B 0,C 180,E1 -6027.564,E2 -6027.564} C_VEL
LIN {X 0,Y 496.005,Z 487.327,A -85,B 0,C 180,E1 -6030,E2 -6030} C_VEL
LIN {X 0,Y 495.832,Z 487.349,A -85,B 0,C 180,E1 -6032.437,E2 -6032.437} C_VEL
LIN {X 0,Y 495.614,Z 487.378,A -85,B 0,C 180,E1 -6034.881,E2 -6034.881} C_VEL
LIN {X 0,Y 495.399,Z 487.494,A -85,B 0,C 180,E1 -6035.7,E2 -6035.7} C_VEL
LIN {X 0,Y 495.382,Z 489.716,A -85,B 0,C 180,E1 -6038.156,E2 -6038.156} C_VEL
LIN {X 0,Y 495.322,Z 493.034,A -85,B 0,C 180,E1 -6041.753,E2 -6041.753} C_VEL
LIN {X 0,Y 495.239,Z 496.203,A -85,B 0,C 180,E1 -6045.202,E2 -6045.202} C_VEL
LIN {X 0,Y 495.148,Z 498.982,A -85,B 0,C 180,E1 -6048.196,E2 -6048.196} C_VEL
LIN {X 0,Y 495.142,Z 500.323,A -85,B 0,C 180,E1 -6049.593,E2 -6049.593} C_VEL
LIN {X 0,Y 499.323,Z 514.559,A -85,B 0,C 180,E1 -6050.08,E2 -6050.08} C_VEL
LIN {X 0,Y 500.555,Z 520.469,A -85,B 0,C 180,E1 -6050.306,E2 -6050.306} C_VEL
LIN {X 0,Y 500.103,Z 534.271,A -85,B 0,C 180,E1 -6050.792,E2 -6050.792} C_VEL
LIN {X 0,Y 499.608,Z 548.449,A -85,B 0,C 180,E1 -6051.453,E2 -6051.453} C_VEL
LIN {X 0,Y 498.956,Z 562.215,A -85,B 0,C 180,E1 -6052.264,E2 -6052.264} C_VEL
LIN {X 0,Y 498.282,Z 575.857,A -85,B 0,C 180,E1 -6053.261,E2 -6053.261} C_VEL
LIN {X 0,Y 497.547,Z 588.672,A -85,B 0,C 180,E1 -6054.404,E2 -6054.404} C_VEL
LIN {X 0,Y 496.984,Z 599.457,A -85,B 0,C 180,E1 -6055.56,E2 -6055.56} C_VEL
LIN {X 0,Y 496.404,Z 610.255,A -85,B 0,C 180,E1 -6056.939,E2 -6056.939} C_VEL
LIN {X 0,Y 496.024,Z 618.522,A -85,B 0,C 180,E1 -6058.194,E2 -6058.194} C_VEL
LIN {X 0,Y 495.624,Z 627.117,A -85,B 0,C 180,E1 -6059.756,E2 -6059.756} C_VEL
LIN {X 0,Y 495.363,Z 633.589,A -85,B 0,C 180,E1 -6061.176,E2 -6061.176} C_VEL
LIN {X 0,Y 495.144,Z 638.997,A -85,B 0,C 180,E1 -6062.64,E2 -6062.64} C_VEL
LIN {X 0,Y 495.051,Z 643.281,A -85,B 0,C 180,E1 -6064.09,E2 -6064.09} C_VEL
LIN {X 0,Y 494.927,Z 646.724,A -85,B 0,C 180,E1 -6065.605,E2 -6065.605} C_VEL
LIN {X 0,Y 494.857,Z 649.349,A -85,B 0,C 180,E1 -6067.314,E2 -6067.314} C_VEL
LIN {X 0,Y 494.856,Z 650.49,A -85,B 0,C 180,E1 -6068.674,E2 -6068.674} C_VEL
LIN {X 0,Y 494.859,Z 650.91,A -85,B 0,C 180,E1 -6069.922,E2 -6069.922} C_VEL
LIN {X 0,Y 494.887,Z 650.232,A -85,B 0,C 180,E1 -6071.871,E2 -6071.871} C_VEL
LIN {X 0,Y 494.941,Z 648.261,A -85,B 0,C 180,E1 -6073.598,E2 -6073.598} C_VEL
LIN {X 0,Y 495.025,Z 645.197,A -85,B 0,C 180,E1 -6075.223,E2 -6075.223} C_VEL
LIN {X 0,Y 495.126,Z 641.315,A -85,B 0,C 180,E1 -6076.719,E2 -6076.719} C_VEL
LIN {X 0,Y 495.285,Z 635.271,A -85,B 0,C 180,E1 -6078.498,E2 -6078.498} C_VEL
LIN {X 0,Y 495.526,Z 628.899,A -85,B 0,C 180,E1 -6079.984,E2 -6079.984} C_VEL
LIN {X 0,Y 495.88,Z 621.443,A -85,B 0,C 180,E1 -6081.42,E2 -6081.42} C_VEL
LIN {X 0,Y 496.326,Z 613.219,A -85,B 0,C 180,E1 -6082.746,E2 -6082.746} C_VEL
LIN {X 0,Y 496.868,Z 602.587,A -85,B 0,C 180,E1 -6084.18,E2 -6084.18} C_VEL
LIN {X 0,Y 497.513,Z 591.088,A -85,B 0,C 180,E1 -6085.465,E2 -6085.465} C_VEL
LIN {X 0,Y 498.198,Z 578.613,A -85,B 0,C 180,E1 -6086.621,E2 -6086.621} C_VEL
LIN {X 0,Y 498.821,Z 565.444,A -85,B 0,C 180,E1 -6087.629,E2 -6087.629} C_VEL
LIN {X 0,Y 499.507,Z 551.133,A -85,B 0,C 180,E1 -6088.51,E2 -6088.51} C_VEL
LIN {X 0,Y 500.093,Z 536.83,A -85,B 0,C 180,E1 -6089.203,E2 -6089.203} C_VEL
LIN {X 0,Y 500.487,Z 522.147,A -85,B 0,C 180,E1 -6089.745,E2 -6089.745} C_VEL
LIN {X 0,Y 500.351,Z 518.715,A -85,B 0,C 180,E1 -6089.852,E2 -6089.852} C_VEL
LIN {X 0,Y 497.17,Z 506.998,A -85,B 0,C 180,E1 -6090.289,E2 -6090.289} C_VEL
LIN {X 0,Y 495.138,Z 500.796,A -85,B 0,C 180,E1 -6090.504,E2 -6090.504} C_VEL
LIN {X 0,Y 495.205,Z 497.829,A -85,B 0,C 180,E1 -6093.899,E2 -6093.899} C_VEL
LIN {X 0,Y 495.238,Z 495.502,A -85,B 0,C 180,E1 -6096.587,E2 -6096.587} C_VEL
LIN {X 0,Y 495.361,Z 493.011,A -85,B 0,C 180,E1 -6099.451,E2 -6099.451} C_VEL
LIN {X 0,Y 495.463,Z 490.96,A -85,B 0,C 180,E1 -6101.872,E2 -6101.872} C_VEL
LIN {X 0,Y 495.53,Z 488.1,A -85,B 0,C 180,E1 -6105.209,E2 -6105.209} C_VEL
LIN {X 0,Y 495.501,Z 487.394,A -85,B 0,C 180,E1 -6106.047,E2 -6106.047} C_VEL
LIN {X 0,Y 495.813,Z 487.353,A -85,B 0,C 180,E1 -6108.554,E2 -6108.554} C_VEL
LIN {X 0,Y 495.87,Z 487.345,A -85,B 0,C 180,E1 -6111.852,E2 -6111.852} C_VEL
LIN {X 0,Y 495.896,Z 487.34,A -85,B 0,C 180,E1 -6114.306,E2 -6114.306} C_VEL
LIN {X 0,Y 495.991,Z 487.33,A -85,B 0,C 180,E1 -6117.563,E2 -6117.563} C_VEL
LIN {X 0,Y 495.994,Z 487.327,A -85,B 0,C 180,E1 -6120,E2 -6120} C_VEL
LIN {X 0,Y 495.989,Z 487.325,A -85,B 0,C 180,E1 -6122.436,E2 -6122.436} C_VEL
LIN {X 0,Y 495.9,Z 487.339,A -85,B 0,C 180,E1 -6125.693,E2 -6125.693} C_VEL
LIN {X 0,Y 495.869,Z 487.34,A -85,B 0,C 180,E1 -6128.148,E2 -6128.148} C_VEL
LIN {X 0,Y 495.851,Z 487.344,A -85,B 0,C 180,E1 -6131.445,E2 -6131.445} C_VEL
LIN {X 0,Y 495.785,Z 487.356,A -85,B 0,C 180,E1 -6134.783,E2 -6134.783} C_VEL
LIN {X 0,Y 495.782,Z 487.351,A -85,B 0,C 180,E1 -6137.318,E2 -6137.318} C_VEL
LIN {X 0,Y 495.773,Z 487.351,A -85,B 0,C 180,E1 -6139.89,E2 -6139.89} C_VEL
LIN {X 0,Y 495.761,Z 487.354,A -85,B 0,C 180,E1 -6142.862,E2 -6142.862} C_VEL
LIN {X 0,Y 495.796,Z 487.354,A -85,B 0,C 180,E1 -6146.067,E2 -6146.067} C_VEL
LIN {X 0,Y 495.777,Z 487.353,A -85,B 0,C 180,E1 -6148.814,E2 -6148.814} C_VEL
LIN {X 0,Y 495.756,Z 487.359,A -85,B 0,C 180,E1 -6151.726,E2 -6151.726} C_VEL
LIN {X 0,Y 495.773,Z 487.352,A -85,B 0,C 180,E1 -6154.695,E2 -6154.695} C_VEL
LIN {X 0,Y 495.729,Z 487.362,A -85,B 0,C 180,E1 -6157.561,E2 -6157.561} C_VEL
LIN {X 0,Y 495.764,Z 487.354,A -85,B 0,C 180,E1 -6160.7,E2 -6160.7} C_VEL
LIN {X 0,Y 495.778,Z 487.536,A -85,B 0,C 180,E1 -6163.857,E2 -6163.857} C_VEL
LIN {X 0,Y 496.771,Z 492.934,A -85,B 0,C 180,E1 -6166.721,E2 -6166.721} C_VEL
LIN {X 0,Y 497.149,Z 496.624,A -85,B 0,C 180,E1 -6168.524,E2 -6168.524} C_VEL
LIN {X 0,Y 496.966,Z 502.319,A -85,B 0,C 180,E1 -6171.059,E2 -6171.059} C_VEL
LIN {X 0,Y 496.699,Z 508.773,A -85,B 0,C 180,E1 -6173.757,E2 -6173.757} C_VEL
LIN {X 0,Y 496.418,Z 516.079,A -85,B 0,C 180,E1 -6176.646,E2 -6176.646} C_VEL
LIN {X 0,Y 496.212,Z 523.225,A -85,B 0,C 180,E1 -6179.344,E2 -6179.344} C_VEL
LIN {X 0,Y 496.004,Z 530.888,A -85,B 0,C 180,E1 -6182.122,E2 -6182.122} C_VEL
LIN {X 0,Y 495.846,Z 538.627,A -85,B 0,C 180,E1 -6184.836,E2 -6184.836} C_VEL
LIN {X 0,Y 495.665,Z 547.728,A -85,B 0,C 180,E1 -6187.93,E2 -6187.93} C_VEL
LIN {X 0,Y 495.604,Z 552.47,A -85,B 0,C 180,E1 -6189.511,E2 -6189.511} C_VEL
LIN {X 0,Y 498.762,Z 566.854,A -85,B 0,C 180,E1 -6189.914,E2 -6189.914} C_VEL
LIN {X 0,Y 500.458,Z 574.745,A -85,B 0,C 180,E1 -6190.188,E2 -6190.188} C_VEL
LIN {X 0,Y 499.955,Z 589.724,A -85,B 0,C 180,E1 -6190.687,E2 -6190.687} C_VEL
LIN {X 0,Y 499.321,Z 605.029,A -85,B 0,C 180,E1 -6191.378,E2 -6191.378} C_VEL
LIN {X 0,Y 498.768,Z 618.477,A -85,B 0,C 180,E1 -6192.153,E2 -6192.153} C_VEL
LIN {X 0,Y 498.122,Z 631.643,A -85,B 0,C 180,E1 -6193.082,E2 -6193.082} C_VEL
LIN {X 0,Y 497.525,Z 644.088,A -85,B 0,C 180,E1 -6194.143,E2 -6194.143} C_VEL
LIN {X 0,Y 496.915,Z 655.087,A -85,B 0,C 180,E1 -6195.251,E2 -6195.251} C_VEL
LIN {X 0,Y 496.439,Z 665.464,A -85,B 0,C 180,E1 -6196.491,E2 -6196.491} C_VEL
LIN {X 0,Y 495.898,Z 675.573,A -85,B 0,C 180,E1 -6197.928,E2 -6197.928} C_VEL
LIN {X 0,Y 495.666,Z 684.057,A -85,B 0,C 180,E1 -6199.378,E2 -6199.378} C_VEL
LIN {X 0,Y 495.354,Z 691.983,A -85,B 0,C 180,E1 -6201.021,E2 -6201.021} C_VEL
LIN {X 0,Y 495.169,Z 698.291,A -85,B 0,C 180,E1 -6202.661,E2 -6202.661} C_VEL
LIN {X 0,Y 495.11,Z 703.174,A -85,B 0,C 180,E1 -6204.297,E2 -6204.297} C_VEL
LIN {X 0,Y 494.992,Z 706.746,A -85,B 0,C 180,E1 -6205.929,E2 -6205.929} C_VEL
LIN {X 0,Y 494.97,Z 709.098,A -85,B 0,C 180,E1 -6207.558,E2 -6207.558} C_VEL
LIN {X 0,Y 494.908,Z 710.278,A -85,B 0,C 180,E1 -6209.186,E2 -6209.186} C_VEL
LIN {X 0,Y 494.908,Z 710.278,A -85,B 0,C 180,E1 -6210.813,E2 -6210.813} C_VEL
LIN {X 0,Y 494.969,Z 709.096,A -85,B 0,C 180,E1 -6212.441,E2 -6212.441} C_VEL
LIN {X 0,Y 494.992,Z 706.747,A -85,B 0,C 180,E1 -6214.07,E2 -6214.07} C_VEL
LIN {X 0,Y 495.107,Z 703.187,A -85,B 0,C 180,E1 -6215.702,E2 -6215.702} C_VEL
LIN {X 0,Y 495.169,Z 698.317,A -85,B 0,C 180,E1 -6217.338,E2 -6217.338} C_VEL
LIN {X 0,Y 495.353,Z 692.016,A -85,B 0,C 180,E1 -6218.978,E2 -6218.978} C_VEL
LIN {X 0,Y 495.665,Z 684.109,A -85,B 0,C 180,E1 -6220.621,E2 -6220.621} C_VEL
LIN {X 0,Y 495.95,Z 675.457,A -85,B 0,C 180,E1 -6222.101,E2 -6222.101} C_VEL
LIN {X 0,Y 496.443,Z 665.578,A -85,B 0,C 180,E1 -6223.508,E2 -6223.508} C_VEL
LIN {X 0,Y 496.906,Z 655.235,A -85,B 0,C 180,E1 -6224.748,E2 -6224.748} C_VEL
LIN {X 0,Y 497.54,Z 643.273,A -85,B 0,C 180,E1 -6225.954,E2 -6225.954} C_VEL
LIN {X 0,Y 498.21,Z 630.574,A -85,B 0,C 180,E1 -6227.019,E2 -6227.019} C_VEL
LIN {X 0,Y 498.91,Z 617.15,A -85,B 0,C 180,E1 -6227.947,E2 -6227.947} C_VEL
LIN {X 0,Y 499.429,Z 604.334,A -85,B 0,C 180,E1 -6228.671,E2 -6228.671} C_VEL
LIN {X 0,Y 500.002,Z 589.944,A -85,B 0,C 180,E1 -6229.315,E2 -6229.315} C_VEL
LIN {X 0,Y 500.472,Z 574.93,A -85,B 0,C 180,E1 -6229.817,E2 -6229.817} C_VEL
LIN {X 0,Y 497.851,Z 562.817,A -85,B 0,C 180,E1 -6230.224,E2 -6230.224} C_VEL
LIN {X 0,Y 495.617,Z 552.902,A -85,B 0,C 180,E1 -6230.497,E2 -6230.497} C_VEL
LIN {X 0,Y 495.823,Z 543.254,A -85,B 0,C 180,E1 -6233.826,E2 -6233.826} C_VEL
LIN {X 0,Y 496.014,Z 534.724,A -85,B 0,C 180,E1 -6236.793,E2 -6236.793} C_VEL
LIN {X 0,Y 496.267,Z 526.684,A -85,B 0,C 180,E1 -6239.712,E2 -6239.712} C_VEL
LIN {X 0,Y 496.501,Z 519.151,A -85,B 0,C 180,E1 -6242.539,E2 -6242.539} C_VEL
LIN {X 0,Y 496.731,Z 511.687,A -85,B 0,C 180,E1 -6245.456,E2 -6245.456} C_VEL
LIN {X 0,Y 497.075,Z 504.277,A -85,B 0,C 180,E1 -6248.469,E2 -6248.469} C_VEL
LIN {X 0,Y 497.365,Z 498.313,A -85,B 0,C 180,E1 -6251.015,E2 -6251.015} C_VEL
LIN {X 0,Y 497.054,Z 494.522,A -85,B 0,C 180,E1 -6252.74,E2 -6252.74} C_VEL
LIN {X 0,Y 496.189,Z 489.668,A -85,B 0,C 180,E1 -6255.087,E2 -6255.087} C_VEL
LIN {X 0,Y 495.764,Z 487.358,A -85,B 0,C 180,E1 -6256.299,E2 -6256.299} C_VEL
LIN {X 0,Y 495.779,Z 487.356,A -85,B 0,C 180,E1 -6259.302,E2 -6259.302} C_VEL
LIN {X 0,Y 495.756,Z 487.358,A -85,B 0,C 180,E1 -6261.409,E2 -6261.409} C_VEL
LIN {X 0,Y 495.749,Z 487.359,A -85,B 0,C 180,E1 -6264.463,E2 -6264.463} C_VEL
LIN {X 0,Y 495.761,Z 487.359,A -85,B 0,C 180,E1 -6267.405,E2 -6267.405} C_VEL
LIN {X 0,Y 495.772,Z 487.355,A -85,B 0,C 180,E1 -6270.254,E2 -6270.254} C_VEL
LIN {X 0,Y 495.824,Z 487.351,A -85,B 0,C 180,E1 -6273.248,E2 -6273.248} C_VEL
LIN {X 0,Y 495.742,Z 487.36,A -85,B 0,C 180,E1 -6275.725,E2 -6275.725} C_VEL
LIN {X 0,Y 495.737,Z 487.36,A -85,B 0,C 180,E1 -6278.371,E2 -6278.371} C_VEL
LIN {X 0,Y 495.775,Z 487.357,A -85,B 0,C 180,E1 -6280.971,E2 -6280.971} C_VEL
LIN {X 0,Y 495.771,Z 487.357,A -85,B 0,C 180,E1 -6283.53,E2 -6283.53} C_VEL
LIN {X 0,Y 495.784,Z 487.356,A -85,B 0,C 180,E1 -6286.056,E2 -6286.056} C_VEL
LIN {X 0,Y 495.859,Z 487.345,A -85,B 0,C 180,E1 -6288.555,E2 -6288.555} C_VEL
LIN {X 0,Y 495.864,Z 487.345,A -85,B 0,C 180,E1 -6291.852,E2 -6291.852} C_VEL
LIN {X 0,Y 495.895,Z 487.339,A -85,B 0,C 180,E1 -6294.307,E2 -6294.307} C_VEL
LIN {X 0,Y 495.985,Z 487.33,A -85,B 0,C 180,E1 -6297.564,E2 -6297.564} C_VEL
LIN {X 0,Y 495.987,Z 487.329,A -85,B 0,C 180,E1 -6300,E2 -6300} C_VEL
LIN {X 0,Y 495.986,Z 487.329,A -85,B 0,C 180,E1 -6302.437,E2 -6302.437} C_VEL
LIN {X 0,Y 495.909,Z 487.34,A -85,B 0,C 180,E1 -6305.694,E2 -6305.694} C_VEL
LIN {X 0,Y 495.864,Z 487.345,A -85,B 0,C 180,E1 -6308.148,E2 -6308.148} C_VEL
LIN {X 0,Y 495.845,Z 487.348,A -85,B 0,C 180,E1 -6311.446,E2 -6311.446} C_VEL
LIN {X 0,Y 495.781,Z 487.354,A -85,B 0,C 180,E1 -6314.784,E2 -6314.784} C_VEL
LIN {X 0,Y 495.78,Z 487.357,A -85,B 0,C 180,E1 -6317.319,E2 -6317.319} C_VEL
LIN {X 0,Y 495.77,Z 487.357,A -85,B 0,C 180,E1 -6319.891,E2 -6319.891} C_VEL
LIN {X 0,Y 495.757,Z 487.358,A -85,B 0,C 180,E1 -6322.863,E2 -6322.863} C_VEL
LIN {X 0,Y 495.792,Z 487.353,A -85,B 0,C 180,E1 -6326.068,E2 -6326.068} C_VEL
LIN {X 0,Y 495.773,Z 487.354,A -85,B 0,C 180,E1 -6328.815,E2 -6328.815} C_VEL
LIN {X 0,Y 495.753,Z 487.359,A -85,B 0,C 180,E1 -6331.727,E2 -6331.727} C_VEL
LIN {X 0,Y 495.771,Z 487.356,A -85,B 0,C 180,E1 -6334.697,E2 -6334.697} C_VEL
LIN {X 0,Y 495.728,Z 487.362,A -85,B 0,C 180,E1 -6337.562,E2 -6337.562} C_VEL
LIN {X 0,Y 495.797,Z 487.354,A -85,B 0,C 180,E1 -6340.054,E2 -6340.054} C_VEL
LIN {X 0,Y 495.76,Z 487.357,A -85,B 0,C 180,E1 -6342.88,E2 -6342.88} C_VEL
LIN {X 0,Y 495.734,Z 487.361,A -85,B 0,C 180,E1 -6346.001,E2 -6346.001} C_VEL
LIN {X 0,Y 495.767,Z 487.355,A -85,B 0,C 180,E1 -6348.706,E2 -6348.706} C_VEL
LIN {X 0,Y 495.763,Z 487.359,A -85,B 0,C 180,E1 -6351.411,E2 -6351.411} C_VEL
LIN {X 0,Y 495.756,Z 487.358,A -85,B 0,C 180,E1 -6354.464,E2 -6354.464} C_VEL
LIN {X 0,Y 495.769,Z 487.357,A -85,B 0,C 180,E1 -6357.407,E2 -6357.407} C_VEL
LIN {X 0,Y 495.767,Z 487.355,A -85,B 0,C 180,E1 -6360.255,E2 -6360.255} C_VEL
LIN {X 0,Y 495.755,Z 487.356,A -85,B 0,C 180,E1 -6360.77,E2 -6360.77} C_VEL
LIN {X 0,Y 495.1,Z 487.441,A -85,B 0,C 180,E1 -6361.449,E2 -6361.449} C_VEL
LIN {X 0,Y 492.247,Z 487.794,A -85,B 0,C 180,E1 -6362.552,E2 -6362.552} C_VEL
LIN {X 0,Y 489.84,Z 488.097,A -85,B 0,C 180,E1 -6363.441,E2 -6363.441} C_VEL
LIN {X 0,Y 488.823,Z 488.222,A -85,B 0,C 180,E1 -6364.127,E2 -6364.127} C_VEL
LIN {X 0,Y 488.75,Z 488.23,A -85,B 0,C 180,E1 -6364.359,E2 -6364.359} C_VEL
LIN {X 0,Y 488.731,Z 488.233,A -85,B 0,C 180,E1 -6367.154,E2 -6367.154} C_VEL
LIN {X 0,Y 488.728,Z 488.235,A -85,B 0,C 180,E1 -6369.811,E2 -6369.811} C_VEL
LIN {X 0,Y 488.738,Z 488.231,A -85,B 0,C 180,E1 -6372.424,E2 -6372.424} C_VEL
LIN {X 0,Y 488.766,Z 488.228,A -85,B 0,C 180,E1 -6375,E2 -6375} C_VEL
LIN {X 0,Y 488.81,Z 488.223,A -85,B 0,C 180,E1 -6378.388,E2 -6378.388} C_VEL
LIN {X 0,Y 488.79,Z 488.227,A -85,B 0,C 180,E1 -6381.734,E2 -6381.734} C_VEL
LIN {X 0,Y 488.86,Z 488.217,A -85,B 0,C 180,E1 -6384.225,E2 -6384.225} C_VEL
LIN {X 0,Y 488.967,Z 488.206,A -85,B 0,C 180,E1 -6387.529,E2 -6387.529} C_VEL
LIN {X 0,Y 488.976,Z 488.203,A -85,B 0,C 180,E1 -6390,E2 -6390} C_VEL
LIN {X 0,Y 488.78,Z 488.227,A -85,B 0,C 180,E1 -6392.473,E2 -6392.473} C_VEL
LIN {X 0,Y 488.55,Z 488.258,A -85,B 0,C 180,E1 -6394.952,E2 -6394.952} C_VEL
LIN {X 0,Y 488.337,Z 488.29,A -85,B 0,C 180,E1 -6395.782,E2 -6395.782} C_VEL
LIN {X 0,Y 488.313,Z 490.542,A -85,B 0,C 180,E1 -6398.275,E2 -6398.275} C_VEL
LIN {X 0,Y 488.263,Z 493.782,A -85,B 0,C 180,E1 -6401.821,E2 -6401.821} C_VEL
LIN {X 0,Y 488.163,Z 496.958,A -85,B 0,C 180,E1 -6405.291,E2 -6405.291} C_VEL
LIN {X 0,Y 488.087,Z 499.907,A -85,B 0,C 180,E1 -6408.468,E2 -6408.468} C_VEL
LIN {X 0,Y 488.064,Z 500.707,A -85,B 0,C 180,E1 -6409.287,E2 -6409.287} C_VEL
LIN {X 0,Y 490.964,Z 509.933,A -85,B 0,C 180,E1 -6409.603,E2 -6409.603} C_VEL
LIN {X 0,Y 493.82,Z 520.919,A -85,B 0,C 180,E1 -6410.03,E2 -6410.03} C_VEL
LIN {X 0,Y 493.411,Z 535.398,A -85,B 0,C 180,E1 -6410.555,E2 -6410.555} C_VEL
LIN {X 0,Y 492.889,Z 549.163,A -85,B 0,C 180,E1 -6411.212,E2 -6411.212} C_VEL
LIN {X 0,Y 492.251,Z 561.895,A -85,B 0,C 180,E1 -6411.969,E2 -6411.969} C_VEL
LIN {X 0,Y 491.511,Z 575.117,A -85,B 0,C 180,E1 -6412.932,E2 -6412.932} C_VEL
LIN {X 0,Y 490.833,Z 587.584,A -85,B 0,C 180,E1 -6414.039,E2 -6414.039} C_VEL
LIN {X 0,Y 490.118,Z 599.284,A -85,B 0,C 180,E1 -6415.287,E2 -6415.287} C_VEL
LIN {X 0,Y 489.532,Z 609.479,A -85,B 0,C 180,E1 -6416.587,E2 -6416.587} C_VEL
LIN {X 0,Y 489.028,Z 619.226,A -85,B 0,C 180,E1 -6418.077,E2 -6418.077} C_VEL
LIN {X 0,Y 488.648,Z 627.056,A -85,B 0,C 180,E1 -6419.512,E2 -6419.512} C_VEL
LIN {X 0,Y 488.356,Z 633.628,A -85,B 0,C 180,E1 -6420.963,E2 -6420.963} C_VEL
LIN {X 0,Y 488.187,Z 638.221,A -85,B 0,C 180,E1 -6422.185,E2 -6422.185} C_VEL
LIN {X 0,Y 488.028,Z 643,A -85,B 0,C 180,E1 -6423.73,E2 -6423.73} C_VEL
LIN {X 0,Y 487.917,Z 646.406,A -85,B 0,C 180,E1 -6425.181,E2 -6425.181} C_VEL
LIN {X 0,Y 487.801,Z 648.299,A -85,B 0,C 180,E1 -6426.213,E2 -6426.213} C_VEL
LIN {X 0,Y 487.786,Z 650.068,A -85,B 0,C 180,E1 -6427.585,E2 -6427.585} C_VEL
LIN {X 0,Y 487.767,Z 651.224,A -85,B 0,C 180,E1 -6429.344,E2 -6429.344} C_VEL
LIN {X 0,Y 487.761,Z 651.291,A -85,B 0,C 180,E1 -6430.42,E2 -6430.42} C_VEL
LIN {X 0,Y 487.787,Z 650.883,A -85,B 0,C 180,E1 -6431.511,E2 -6431.511} C_VEL
LIN {X 0,Y 487.832,Z 649.895,A -85,B 0,C 180,E1 -6432.714,E2 -6432.714} C_VEL
LIN {X 0,Y 487.873,Z 648.256,A -85,B 0,C 180,E1 -6433.923,E2 -6433.923} C_VEL
LIN {X 0,Y 487.971,Z 644.926,A -85,B 0,C 180,E1 -6435.618,E2 -6435.618} C_VEL
LIN {X 0,Y 488.126,Z 639.957,A -85,B 0,C 180,E1 -6437.413,E2 -6437.413} C_VEL
LIN {X 0,Y 488.333,Z 633.88,A -85,B 0,C 180,E1 -6439.093,E2 -6439.093} C_VEL
LIN {X 0,Y 488.693,Z 626.359,A -85,B 0,C 180,E1 -6440.744,E2 -6440.744} C_VEL
LIN {X 0,Y 489.16,Z 617.12,A -85,B 0,C 180,E1 -6442.386,E2 -6442.386} C_VEL
LIN {X 0,Y 489.64,Z 608.035,A -85,B 0,C 180,E1 -6443.731,E2 -6443.731} C_VEL
LIN {X 0,Y 490.265,Z 597.729,A -85,B 0,C 180,E1 -6445.012,E2 -6445.012} C_VEL
LIN {X 0,Y 490.963,Z 586.05,A -85,B 0,C 180,E1 -6446.226,E2 -6446.226} C_VEL
LIN {X 0,Y 491.65,Z 573.289,A -85,B 0,C 180,E1 -6447.329,E2 -6447.329} C_VEL
LIN {X 0,Y 492.363,Z 560.743,A -85,B 0,C 180,E1 -6448.217,E2 -6448.217} C_VEL
LIN {X 0,Y 492.992,Z 546.617,A -85,B 0,C 180,E1 -6449.032,E2 -6449.032} C_VEL
LIN {X 0,Y 493.581,Z 531.533,A -85,B 0,C 180,E1 -6449.705,E2 -6449.705} C_VEL
LIN {X 0,Y 493.722,Z 520.414,A -85,B 0,C 180,E1 -6450.089,E2 -6450.089} C_VEL
LIN {X 0,Y 490.663,Z 509.007,A -85,B 0,C 180,E1 -6450.533,E2 -6450.533} C_VEL
LIN {X 0,Y 488.091,Z 501.288,A -85,B 0,C 180,E1 -6450.818,E2 -6450.818} C_VEL
LIN {X 0,Y 488.151,Z 498.94,A -85,B 0,C 180,E1 -6453.492,E2 -6453.492} C_VEL
LIN {X 0,Y 488.205,Z 496.589,A -85,B 0,C 180,E1 -6456.229,E2 -6456.229} C_VEL
LIN {X 0,Y 488.311,Z 493.941,A -85,B 0,C 180,E1 -6459.309,E2 -6459.309} C_VEL
LIN {X 0,Y 488.415,Z 491.346,A -85,B 0,C 180,E1 -6462.411,E2 -6462.411} C_VEL
LIN {X 0,Y 488.481,Z 489.15,A -85,B 0,C 180,E1 -6464.99,E2 -6464.99} C_VEL
LIN {X 0,Y 488.451,Z 488.426,A -85,B 0,C 180,E1 -6465.841,E2 -6465.841} C_VEL
LIN {X 0,Y 488.75,Z 488.235,A -85,B 0,C 180,E1 -6468.386,E2 -6468.386} C_VEL
LIN {X 0,Y 488.815,Z 488.223,A -85,B 0,C 180,E1 -6471.733,E2 -6471.733} C_VEL
LIN {X 0,Y 488.855,Z 488.218,A -85,B 0,C 180,E1 -6474.224,E2 -6474.224} C_VEL
LIN {X 0,Y 488.958,Z 488.205,A -85,B 0,C 180,E1 -6477.528,E2 -6477.528} C_VEL
LIN {X 0,Y 488.951,Z 488.202,A -85,B 0,C 180,E1 -6480.823,E2 -6480.823} C_VEL
LIN {X 0,Y 488.957,Z 488.201,A -85,B 0,C 180,E1 -6482.471,E2 -6482.471} C_VEL
LIN {X 0,Y 488.858,Z 488.215,A -85,B 0,C 180,E1 -6485.775,E2 -6485.775} C_VEL
LIN {X 0,Y 488.814,Z 488.219,A -85,B 0,C 180,E1 -6488.266,E2 -6488.266} C_VEL
LIN {X 0,Y 488.804,Z 488.22,A -85,B 0,C 180,E1 -6491.612,E2 -6491.612} C_VEL
LIN {X 0,Y 488.757,Z 488.229,A -85,B 0,C 180,E1 -6495,E2 -6495} C_VEL
LIN {X 0,Y 488.751,Z 488.231,A -85,B 0,C 180,E1 -6498.442,E2 -6498.442} C_VEL
LIN {X 0,Y 488.703,Z 488.233,A -85,B 0,C 180,E1 -6501.071,E2 -6501.071} C_VEL
LIN {X 0,Y 488.69,Z 488.234,A -85,B 0,C 180,E1 -6503.745,E2 -6503.745} C_VEL
LIN {X 0,Y 488.795,Z 488.221,A -85,B 0,C 180,E1 -6506.945,E2 -6506.945} C_VEL
LIN {X 0,Y 488.716,Z 488.235,A -85,B 0,C 180,E1 -6510.365,E2 -6510.365} C_VEL
LIN {X 0,Y 488.733,Z 488.233,A -85,B 0,C 180,E1 -6513.485,E2 -6513.485} C_VEL
LIN {X 0,Y 488.686,Z 488.237,A -85,B 0,C 180,E1 -6516.356,E2 -6516.356} C_VEL
LIN {X 0,Y 488.699,Z 488.231,A -85,B 0,C 180,E1 -6519.254,E2 -6519.254} C_VEL
LIN {X 0,Y 488.721,Z 488.234,A -85,B 0,C 180,E1 -6521.602,E2 -6521.602} C_VEL
LIN {X 0,Y 488.712,Z 488.291,A -85,B 0,C 180,E1 -6523.426,E2 -6523.426} C_VEL
LIN {X 0,Y 489.72,Z 493.854,A -85,B 0,C 180,E1 -6526.461,E2 -6526.461} C_VEL
LIN {X 0,Y 490.181,Z 497.373,A -85,B 0,C 180,E1 -6528.206,E2 -6528.206} C_VEL
LIN {X 0,Y 490.034,Z 501.972,A -85,B 0,C 180,E1 -6530.329,E2 -6530.329} C_VEL
LIN {X 0,Y 489.766,Z 507.977,A -85,B 0,C 180,E1 -6532.938,E2 -6532.938} C_VEL
LIN {X 0,Y 489.504,Z 515.365,A -85,B 0,C 180,E1 -6535.949,E2 -6535.949} C_VEL
LIN {X 0,Y 489.263,Z 522.871,A -85,B 0,C 180,E1 -6538.861,E2 -6538.861} C_VEL
LIN {X 0,Y 488.95,Z 531.77,A -85,B 0,C 180,E1 -6542.151,E2 -6542.151} C_VEL
LIN {X 0,Y 488.759,Z 539.589,A -85,B 0,C 180,E1 -6544.944,E2 -6544.944} C_VEL
LIN {X 0,Y 488.571,Z 548.514,A -85,B 0,C 180,E1 -6548.037,E2 -6548.037} C_VEL
LIN {X 0,Y 488.541,Z 551.924,A -85,B 0,C 180,E1 -6549.198,E2 -6549.198} C_VEL
LIN {X 0,Y 492.079,Z 568.219,A -85,B 0,C 180,E1 -6549.676,E2 -6549.676} C_VEL
LIN {X 0,Y 493.691,Z 575.946,A -85,B 0,C 180,E1 -6549.958,E2 -6549.958} C_VEL
LIN {X 0,Y 493.168,Z 590.986,A -85,B 0,C 180,E1 -6550.487,E2 -6550.487} C_VEL
LIN {X 0,Y 492.495,Z 605.478,A -85,B 0,C 180,E1 -6551.164,E2 -6551.164} C_VEL
LIN {X 0,Y 491.843,Z 619.533,A -85,B 0,C 180,E1 -6552.001,E2 -6552.001} C_VEL
LIN {X 0,Y 491.169,Z 632.42,A -85,B 0,C 180,E1 -6552.943,E2 -6552.943} C_VEL
LIN {X 0,Y 490.509,Z 645.277,A -85,B 0,C 180,E1 -6554.078,E2 -6554.078} C_VEL
LIN {X 0,Y 489.855,Z 656.389,A -85,B 0,C 180,E1 -6555.246,E2 -6555.246} C_VEL
LIN {X 0,Y 489.351,Z 666.511,A -85,B 0,C 180,E1 -6556.504,E2 -6556.504} C_VEL
LIN {X 0,Y 488.826,Z 675.8,A -85,B 0,C 180,E1 -6557.865,E2 -6557.865} C_VEL
LIN {X 0,Y 488.547,Z 684.687,A -85,B 0,C 180,E1 -6559.431,E2 -6559.431} C_VEL
LIN {X 0,Y 488.279,Z 691.519,A -85,B 0,C 180,E1 -6560.89,E2 -6560.89} C_VEL
LIN {X 0,Y 488.079,Z 697.836,A -85,B 0,C 180,E1 -6562.554,E2 -6562.554} C_VEL
LIN {X 0,Y 488.004,Z 702.726,A -85,B 0,C 180,E1 -6564.214,E2 -6564.214} C_VEL
LIN {X 0,Y 487.897,Z 706.306,A -85,B 0,C 180,E1 -6565.869,E2 -6565.869} C_VEL
LIN {X 0,Y 487.882,Z 708.665,A -85,B 0,C 180,E1 -6567.523,E2 -6567.523} C_VEL
LIN {X 0,Y 487.831,Z 709.851,A -85,B 0,C 180,E1 -6569.174,E2 -6569.174} C_VEL
LIN {X 0,Y 487.831,Z 709.854,A -85,B 0,C 180,E1 -6570.825,E2 -6570.825} C_VEL
LIN {X 0,Y 487.882,Z 708.672,A -85,B 0,C 180,E1 -6572.476,E2 -6572.476} C_VEL
LIN {X 0,Y 487.896,Z 706.324,A -85,B 0,C 180,E1 -6574.13,E2 -6574.13} C_VEL
LIN {X 0,Y 488.002,Z 702.763,A -85,B 0,C 180,E1 -6575.785,E2 -6575.785} C_VEL
LIN {X 0,Y 488.078,Z 697.892,A -85,B 0,C 180,E1 -6577.446,E2 -6577.446} C_VEL
LIN {X 0,Y 488.279,Z 691.59,A -85,B 0,C 180,E1 -6579.109,E2 -6579.109} C_VEL
LIN {X 0,Y 488.635,Z 683.681,A -85,B 0,C 180,E1 -6580.776,E2 -6580.776} C_VEL
LIN {X 0,Y 488.889,Z 675.716,A -85,B 0,C 180,E1 -6582.169,E2 -6582.169} C_VEL
LIN {X 0,Y 489.451,Z 665.141,A -85,B 0,C 180,E1 -6583.704,E2 -6583.704} C_VEL
LIN {X 0,Y 489.945,Z 654.796,A -85,B 0,C 180,E1 -6584.963,E2 -6584.963} C_VEL
LIN {X 0,Y 490.627,Z 642.734,A -85,B 0,C 180,E1 -6586.194,E2 -6586.194} C_VEL
LIN {X 0,Y 491.349,Z 630.129,A -85,B 0,C 180,E1 -6587.265,E2 -6587.265} C_VEL
LIN {X 0,Y 492.055,Z 616.699,A -85,B 0,C 180,E1 -6588.206,E2 -6588.206} C_VEL
LIN {X 0,Y 492.737,Z 601.895,A -85,B 0,C 180,E1 -6589.042,E2 -6589.042} C_VEL
LIN {X 0,Y 493.367,Z 586.701,A -85,B 0,C 180,E1 -6589.702,E2 -6589.702} C_VEL
LIN {X 0,Y 493.6,Z 574.969,A -85,B 0,C 180,E1 -6590.089,E2 -6590.089} C_VEL
LIN {X 0,Y 489.932,Z 558.934,A -85,B 0,C 180,E1 -6590.627,E2 -6590.627} C_VEL
LIN {X 0,Y 488.559,Z 552.448,A -85,B 0,C 180,E1 -6590.823,E2 -6590.823} C_VEL
LIN {X 0,Y 488.761,Z 544.112,A -85,B 0,C 180,E1 -6593.741,E2 -6593.741} C_VEL
LIN {X 0,Y 488.954,Z 536.445,A -85,B 0,C 180,E1 -6596.459,E2 -6596.459} C_VEL
LIN {X 0,Y 489.238,Z 527.653,A -85,B 0,C 180,E1 -6599.708,E2 -6599.708} C_VEL
LIN {X 0,Y 489.476,Z 520.127,A -85,B 0,C 180,E1 -6602.576,E2 -6602.576} C_VEL
LIN {X 0,Y 489.726,Z 512.675,A -85,B 0,C 180,E1 -6605.534,E2 -6605.534} C_VEL
LIN {X 0,Y 490.1,Z 505.301,A -85,B 0,C 180,E1 -6608.592,E2 -6608.592} C_VEL
LIN {X 0,Y 490.387,Z 499.189,A -85,B 0,C 180,E1 -6611.241,E2 -6611.241} C_VEL
LIN {X 0,Y 489.854,Z 494.317,A -85,B 0,C 180,E1 -6613.523,E2 -6613.523} C_VEL
LIN {X 0,Y 488.711,Z 488.237,A -85,B 0,C 180,E1 -6616.628,E2 -6616.628} C_VEL
LIN {X 0,Y 488.762,Z 488.231,A -85,B 0,C 180,E1 -6619.68,E2 -6619.68} C_VEL
LIN {X 0,Y 488.675,Z 488.241,A -85,B 0,C 180,E1 -6622.841,E2 -6622.841} C_VEL
LIN {X 0,Y 488.727,Z 488.234,A -85,B 0,C 180,E1 -6625.887,E2 -6625.887} C_VEL
LIN {X 0,Y 488.687,Z 488.239,A -85,B 0,C 180,E1 -6628.82,E2 -6628.82} C_VEL
LIN {X 0,Y 488.737,Z 488.234,A -85,B 0,C 180,E1 -6631.671,E2 -6631.671} C_VEL
LIN {X 0,Y 488.741,Z 488.23,A -85,B 0,C 180,E1 -6634.444,E2 -6634.444} C_VEL
LIN {X 0,Y 488.71,Z 488.236,A -85,B 0,C 180,E1 -6637.153,E2 -6637.153} C_VEL
LIN {X 0,Y 488.718,Z 488.235,A -85,B 0,C 180,E1 -6639.81,E2 -6639.81} C_VEL
LIN {X 0,Y 488.725,Z 488.232,A -85,B 0,C 180,E1 -6642.423,E2 -6642.423} C_VEL
LIN {X 0,Y 488.751,Z 488.23,A -85,B 0,C 180,E1 -6645,E2 -6645} C_VEL
LIN {X 0,Y 488.82,Z 488.221,A -85,B 0,C 180,E1 -6648.388,E2 -6648.388} C_VEL
LIN {X 0,Y 488.809,Z 488.225,A -85,B 0,C 180,E1 -6651.734,E2 -6651.734} C_VEL
LIN {X 0,Y 488.853,Z 488.216,A -85,B 0,C 180,E1 -6654.225,E2 -6654.225} C_VEL
LIN {X 0,Y 488.953,Z 488.207,A -85,B 0,C 180,E1 -6657.529,E2 -6657.529} C_VEL
LIN {X 0,Y 488.959,Z 488.205,A -85,B 0,C 180,E1 -6660,E2 -6660} C_VEL
LIN {X 0,Y 488.954,Z 488.204,A -85,B 0,C 180,E1 -6662.472,E2 -6662.472} C_VEL
LIN {X 0,Y 488.865,Z 488.218,A -85,B 0,C 180,E1 -6665.776,E2 -6665.776} C_VEL
LIN {X 0,Y 488.809,Z 488.223,A -85,B 0,C 180,E1 -6668.267,E2 -6668.267} C_VEL
LIN {X 0,Y 488.798,Z 488.227,A -85,B 0,C 180,E1 -6671.613,E2 -6671.613} C_VEL
LIN {X 0,Y 488.752,Z 488.231,A -85,B 0,C 180,E1 -6675.001,E2 -6675.001} C_VEL
LIN {X 0,Y 488.746,Z 488.23,A -85,B 0,C 180,E1 -6678.443,E2 -6678.443} C_VEL
LIN {X 0,Y 488.698,Z 488.237,A -85,B 0,C 180,E1 -6681.072,E2 -6681.072} C_VEL
LIN {X 0,Y 488.686,Z 488.24,A -85,B 0,C 180,E1 -6683.746,E2 -6683.746} C_VEL
LIN {X 0,Y 488.792,Z 488.225,A -85,B 0,C 180,E1 -6686.946,E2 -6686.946} C_VEL
LIN {X 0,Y 488.712,Z 488.235,A -85,B 0,C 180,E1 -6690.366,E2 -6690.366} C_VEL
LIN {X 0,Y 488.73,Z 488.235,A -85,B 0,C 180,E1 -6693.486,E2 -6693.486} C_VEL
LIN {X 0,Y 488.684,Z 488.238,A -85,B 0,C 180,E1 -6696.357,E2 -6696.357} C_VEL
LIN {X 0,Y 488.745,Z 488.233,A -85,B 0,C 180,E1 -6699.251,E2 -6699.251} C_VEL
LIN {X 0,Y 488.729,Z 488.234,A -85,B 0,C 180,E1 -6701.604,E2 -6701.604} C_VEL
LIN {X 0,Y 488.699,Z 488.237,A -85,B 0,C 180,E1 -6704.025,E2 -6704.025} C_VEL
LIN {X 0,Y 488.741,Z 488.233,A -85,B 0,C 180,E1 -6707.17,E2 -6707.17} C_VEL
LIN {X 0,Y 488.734,Z 488.233,A -85,B 0,C 180,E1 -6709.678,E2 -6709.678} C_VEL
LIN {X 0,Y 488.682,Z 488.239,A -85,B 0,C 180,E1 -6712.278,E2 -6712.278} C_VEL
LIN {X 0,Y 488.727,Z 488.233,A -85,B 0,C 180,E1 -6715.053,E2 -6715.053} C_VEL
LIN {X 0,Y 488.705,Z 488.236,A -85,B 0,C 180,E1 -6718.047,E2 -6718.047} C_VEL
LIN {X 0,Y 488.724,Z 488.232,A -85,B 0,C 180,E1 -6720.768,E2 -6720.768} C_VEL
LIN {X 0,Y 488.769,Z 488.23,A -85,B 0,C 180,E1 -6723.53,E2 -6723.53} C_VEL
LIN {X 0,Y 488.75,Z 488.23,A -85,B 0,C 180,E1 -6724.359,E2 -6724.359} C_VEL
LIN {X 0,Y 488.103,Z 488.313,A -85,B 0,C 180,E1 -6725.047,E2 -6725.047} C_VEL
LIN {X 0,Y 485.234,Z 488.674,A -85,B 0,C 180,E1 -6726.163,E2 -6726.163} C_VEL
LIN {X 0,Y 482.788,Z 488.978,A -85,B 0,C 180,E1 -6727.063,E2 -6727.063} C_VEL
LIN {X 0,Y 481.73,Z 489.107,A -85,B 0,C 180,E1 -6727.759,E2 -6727.759} C_VEL
LIN {X 0,Y 481.641,Z 489.116,A -85,B 0,C 180,E1 -6727.994,E2 -6727.994} C_VEL
LIN {X 0,Y 481.709,Z 489.106,A -85,B 0,C 180,E1 -6730.394,E2 -6730.394} C_VEL
LIN {X 0,Y 481.695,Z 489.108,A -85,B 0,C 180,E1 -6733.035,E2 -6733.035} C_VEL
LIN {X 0,Y 481.694,Z 489.111,A -85,B 0,C 180,E1 -6735.64,E2 -6735.64} C_VEL
LIN {X 0,Y 481.755,Z 489.101,A -85,B 0,C 180,E1 -6738.216,E2 -6738.216} C_VEL
LIN {X 0,Y 481.744,Z 489.104,A -85,B 0,C 180,E1 -6741.612,E2 -6741.612} C_VEL
LIN {X 0,Y 481.821,Z 489.094,A -85,B 0,C 180,E1 -6744.14,E2 -6744.14} C_VEL
LIN {X 0,Y 481.934,Z 489.081,A -85,B 0,C 180,E1 -6747.493,E2 -6747.493} C_VEL
LIN {X 0,Y 481.947,Z 489.078,A -85,B 0,C 180,E1 -6750,E2 -6750} C_VEL
LIN {X 0,Y 481.731,Z 489.105,A -85,B 0,C 180,E1 -6752.509,E2 -6752.509} C_VEL
LIN {X 0,Y 481.49,Z 489.137,A -85,B 0,C 180,E1 -6755.025,E2 -6755.025} C_VEL
LIN {X 0,Y 481.282,Z 489.163,A -85,B 0,C 180,E1 -6755.867,E2 -6755.867} C_VEL
LIN {X 0,Y 481.261,Z 491.366,A -85,B 0,C 180,E1 -6758.397,E2 -6758.397} C_VEL
LIN {X 0,Y 481.192,Z 494.506,A -85,B 0,C 180,E1 -6761.883,E2 -6761.883} C_VEL
LIN {X 0,Y 481.088,Z 497.746,A -85,B 0,C 180,E1 -6765.383,E2 -6765.383} C_VEL
LIN {X 0,Y 481.03,Z 501.02,A -85,B 0,C 180,E1 -6768.948,E2 -6768.948} C_VEL
LIN {X 0,Y 483.04,Z 507.535,A -85,B 0,C 180,E1 -6769.186,E2 -6769.186} C_VEL
LIN {X 0,Y 486.297,Z 518.611,A -85,B 0,C 180,E1 -6769.626,E2 -6769.626} C_VEL
LIN {X 0,Y 487.174,Z 523.433,A -85,B 0,C 180,E1 -6769.815,E2 -6769.815} C_VEL
LIN {X 0,Y 486.651,Z 538.389,A -85,B 0,C 180,E1 -6770.39,E2 -6770.39} C_VEL
LIN {X 0,Y 486.018,Z 552.124,A -85,B 0,C 180,E1 -6771.082,E2 -6771.082} C_VEL
LIN {X 0,Y 485.312,Z 565.333,A -85,B 0,C 180,E1 -6771.917,E2 -6771.917} C_VEL
LIN {X 0,Y 484.621,Z 578.493,A -85,B 0,C 180,E1 -6772.939,E2 -6772.939} C_VEL
LIN {X 0,Y 483.769,Z 591.048,A -85,B 0,C 180,E1 -6774.116,E2 -6774.116} C_VEL
LIN {X 0,Y 483.118,Z 601.675,A -85,B 0,C 180,E1 -6775.316,E2 -6775.316} C_VEL
LIN {X 0,Y 482.532,Z 611.355,A -85,B 0,C 180,E1 -6776.607,E2 -6776.607} C_VEL
LIN {X 0,Y 482,Z 620.459,A -85,B 0,C 180,E1 -6778.049,E2 -6778.049} C_VEL
LIN {X 0,Y 481.537,Z 629.3,A -85,B 0,C 180,E1 -6779.751,E2 -6779.751} C_VEL
LIN {X 0,Y 481.25,Z 635.569,A -85,B 0,C 180,E1 -6781.227,E2 -6781.227} C_VEL
LIN {X 0,Y 481.016,Z 640.791,A -85,B 0,C 180,E1 -6782.724,E2 -6782.724} C_VEL
LIN {X 0,Y 480.895,Z 644.91,A -85,B 0,C 180,E1 -6784.239,E2 -6784.239} C_VEL
LIN {X 0,Y 480.763,Z 648.078,A -85,B 0,C 180,E1 -6785.784,E2 -6785.784} C_VEL
LIN {X 0,Y 480.695,Z 649.658,A -85,B 0,C 180,E1 -6786.83,E2 -6786.83} C_VEL
LIN {X 0,Y 480.705,Z 650.802,A -85,B 0,C 180,E1 -6787.883,E2 -6787.883} C_VEL
LIN {X 0,Y 480.676,Z 651.625,A -85,B 0,C 180,E1 -6789.202,E2 -6789.202} C_VEL
LIN {X 0,Y 480.672,Z 651.702,A -85,B 0,C 180,E1 -6790.508,E2 -6790.508} C_VEL
LIN {X 0,Y 480.71,Z 650.782,A -85,B 0,C 180,E1 -6792.262,E2 -6792.262} C_VEL
LIN {X 0,Y 480.784,Z 649.523,A -85,B 0,C 180,E1 -6793.396,E2 -6793.396} C_VEL
LIN {X 0,Y 480.817,Z 647.715,A -85,B 0,C 180,E1 -6794.555,E2 -6794.555} C_VEL
LIN {X 0,Y 480.931,Z 644.175,A -85,B 0,C 180,E1 -6796.177,E2 -6796.177} C_VEL
LIN {X 0,Y 481.121,Z 639.525,A -85,B 0,C 180,E1 -6797.782,E2 -6797.782} C_VEL
LIN {X 0,Y 481.323,Z 633.583,A -85,B 0,C 180,E1 -6799.4,E2 -6799.4} C_VEL
LIN {X 0,Y 481.708,Z 626.786,A -85,B 0,C 180,E1 -6800.902,E2 -6800.902} C_VEL
LIN {X 0,Y 482.185,Z 617.883,A -85,B 0,C 180,E1 -6802.513,E2 -6802.513} C_VEL
LIN {X 0,Y 482.717,Z 608.924,A -85,B 0,C 180,E1 -6803.867,E2 -6803.867} C_VEL
LIN {X 0,Y 483.392,Z 598.361,A -85,B 0,C 180,E1 -6805.204,E2 -6805.204} C_VEL
LIN {X 0,Y 484.123,Z 586.907,A -85,B 0,C 180,E1 -6806.415,E2 -6806.415} C_VEL
LIN {X 0,Y 484.887,Z 573.805,A -85,B 0,C 180,E1 -6807.569,E2 -6807.569} C_VEL
LIN {X 0,Y 485.655,Z 561.09,A -85,B 0,C 180,E1 -6808.481,E2 -6808.481} C_VEL
LIN {X 0,Y 486.312,Z 546.81,A -85,B 0,C 180,E1 -6809.314,E2 -6809.314} C_VEL
LIN {X 0,Y 486.922,Z 531.632,A -85,B 0,C 180,E1 -6809.997,E2 -6809.997} C_VEL
LIN {X 0,Y 487.034,Z 521.651,A -85,B 0,C 180,E1 -6810.35,E2 -6810.35} C_VEL
LIN {X 0,Y 484.3,Z 511.423,A -85,B 0,C 180,E1 -6810.764,E2 -6810.764} C_VEL
LIN {X 0,Y 481.046,Z 501.774,A -85,B 0,C 180,E1 -6811.131,E2 -6811.131} C_VEL
LIN {X 0,Y 481.08,Z 499.287,A -85,B 0,C 180,E1 -6814.006,E2 -6814.006} C_VEL
LIN {X 0,Y 481.162,Z 496.764,A -85,B 0,C 180,E1 -6816.953,E2 -6816.953} C_VEL
LIN {X 0,Y 481.279,Z 494.633,A -85,B 0,C 180,E1 -6819.484,E2 -6819.484} C_VEL
LIN {X 0,Y 481.352,Z 492.391,A -85,B 0,C 180,E1 -6822.144,E2 -6822.144} C_VEL
LIN {X 0,Y 481.425,Z 490.204,A -85,B 0,C 180,E1 -6824.765,E2 -6824.765} C_VEL
LIN {X 0,Y 481.459,Z 489.142,A -85,B 0,C 180,E1 -6826.493,E2 -6826.493} C_VEL
LIN {X 0,Y 481.685,Z 489.11,A -85,B 0,C 180,E1 -6829.066,E2 -6829.066} C_VEL
LIN {X 0,Y 481.825,Z 489.092,A -85,B 0,C 180,E1 -6832.456,E2 -6832.456} C_VEL
LIN {X 0,Y 481.782,Z 489.095,A -85,B 0,C 180,E1 -6834.978,E2 -6834.978} C_VEL
LIN {X 0,Y 481.925,Z 489.081,A -85,B 0,C 180,E1 -6837.492,E2 -6837.492} C_VEL
LIN {X 0,Y 481.902,Z 489.081,A -85,B 0,C 180,E1 -6840.835,E2 -6840.835} C_VEL
LIN {X 0,Y 481.924,Z 489.077,A -85,B 0,C 180,E1 -6842.507,E2 -6842.507} C_VEL
LIN {X 0,Y 481.818,Z 489.092,A -85,B 0,C 180,E1 -6845.86,E2 -6845.86} C_VEL
LIN {X 0,Y 481.759,Z 489.098,A -85,B 0,C 180,E1 -6848.388,E2 -6848.388} C_VEL
LIN {X 0,Y 481.748,Z 489.099,A -85,B 0,C 180,E1 -6851.785,E2 -6851.785} C_VEL
LIN {X 0,Y 481.738,Z 489.102,A -85,B 0,C 180,E1 -6855.224,E2 -6855.224} C_VEL
LIN {X 0,Y 481.708,Z 489.108,A -85,B 0,C 180,E1 -6858.722,E2 -6858.722} C_VEL
LIN {X 0,Y 481.643,Z 489.111,A -85,B 0,C 180,E1 -6861.395,E2 -6861.395} C_VEL
LIN {X 0,Y 481.674,Z 489.112,A -85,B 0,C 180,E1 -6864.113,E2 -6864.113} C_VEL
LIN {X 0,Y 481.748,Z 489.099,A -85,B 0,C 180,E1 -6867.141,E2 -6867.141} C_VEL
LIN {X 0,Y 481.685,Z 489.112,A -85,B 0,C 180,E1 -6869.74,E2 -6869.74} C_VEL
LIN {X 0,Y 481.67,Z 489.11,A -85,B 0,C 180,E1 -6872.674,E2 -6872.674} C_VEL
LIN {X 0,Y 481.64,Z 489.117,A -85,B 0,C 180,E1 -6875.709,E2 -6875.709} C_VEL
LIN {X 0,Y 481.668,Z 489.107,A -85,B 0,C 180,E1 -6878.859,E2 -6878.859} C_VEL
LIN {X 0,Y 481.66,Z 489.115,A -85,B 0,C 180,E1 -6881.914,E2 -6881.914} C_VEL
LIN {X 0,Y 481.694,Z 489.222,A -85,B 0,C 180,E1 -6883.079,E2 -6883.079} C_VEL
LIN {X 0,Y 482.67,Z 494.668,A -85,B 0,C 180,E1 -6886.12,E2 -6886.12} C_VEL
LIN {X 0,Y 483.195,Z 498.296,A -85,B 0,C 180,E1 -6888.006,E2 -6888.006} C_VEL
LIN {X 0,Y 483.047,Z 503.517,A -85,B 0,C 180,E1 -6890.454,E2 -6890.454} C_VEL
LIN {X 0,Y 482.703,Z 510.143,A -85,B 0,C 180,E1 -6893.349,E2 -6893.349} C_VEL
LIN {X 0,Y 482.459,Z 516.873,A -85,B 0,C 180,E1 -6896.131,E2 -6896.131} C_VEL
LIN {X 0,Y 482.244,Z 523.774,A -85,B 0,C 180,E1 -6898.845,E2 -6898.845} C_VEL
LIN {X 0,Y 481.895,Z 532.635,A -85,B 0,C 180,E1 -6902.18,E2 -6902.18} C_VEL
LIN {X 0,Y 481.683,Z 540.32,A -85,B 0,C 180,E1 -6904.968,E2 -6904.968} C_VEL
LIN {X 0,Y 481.511,Z 549.329,A -85,B 0,C 180,E1 -6908.149,E2 -6908.149} C_VEL
LIN {X 0,Y 481.496,Z 551.425,A -85,B 0,C 180,E1 -6908.879,E2 -6908.879} C_VEL
LIN {X 0,Y 485.065,Z 568.256,A -85,B 0,C 180,E1 -6909.385,E2 -6909.385} C_VEL
LIN {X 0,Y 486.951,Z 576.799,A -85,B 0,C 180,E1 -6909.711,E2 -6909.711} C_VEL
LIN {X 0,Y 486.376,Z 592.462,A -85,B 0,C 180,E1 -6910.289,E2 -6910.289} C_VEL
LIN {X 0,Y 485.66,Z 606.927,A -85,B 0,C 180,E1 -6910.998,E2 -6910.998} C_VEL
LIN {X 0,Y 484.926,Z 620.588,A -85,B 0,C 180,E1 -6911.844,E2 -6911.844} C_VEL
LIN {X 0,Y 484.141,Z 634.504,A -85,B 0,C 180,E1 -6912.905,E2 -6912.905} C_VEL
LIN {X 0,Y 483.442,Z 647.116,A -85,B 0,C 180,E1 -6914.074,E2 -6914.074} C_VEL
LIN {X 0,Y 482.783,Z 657.695,A -85,B 0,C 180,E1 -6915.241,E2 -6915.241} C_VEL
LIN {X 0,Y 482.273,Z 667.526,A -85,B 0,C 180,E1 -6916.516,E2 -6916.516} C_VEL
LIN {X 0,Y 481.752,Z 676.882,A -85,B 0,C 180,E1 -6917.95,E2 -6917.95} C_VEL
LIN {X 0,Y 481.432,Z 685.24,A -85,B 0,C 180,E1 -6919.486,E2 -6919.486} C_VEL
LIN {X 0,Y 481.144,Z 692.76,A -85,B 0,C 180,E1 -6921.177,E2 -6921.177} C_VEL
LIN {X 0,Y 480.988,Z 698.732,A -85,B 0,C 180,E1 -6922.865,E2 -6922.865} C_VEL
LIN {X 0,Y 480.907,Z 702.279,A -85,B 0,C 180,E1 -6924.128,E2 -6924.128} C_VEL
LIN {X 0,Y 480.804,Z 705.866,A -85,B 0,C 180,E1 -6925.808,E2 -6925.808} C_VEL
LIN {X 0,Y 480.798,Z 708.232,A -85,B 0,C 180,E1 -6927.486,E2 -6927.486} C_VEL
LIN {X 0,Y 480.757,Z 709.424,A -85,B 0,C 180,E1 -6929.162,E2 -6929.162} C_VEL
LIN {X 0,Y 480.757,Z 709.43,A -85,B 0,C 180,E1 -6930.837,E2 -6930.837} C_VEL
LIN {X 0,Y 480.798,Z 708.249,A -85,B 0,C 180,E1 -6932.513,E2 -6932.513} C_VEL
LIN {X 0,Y 480.802,Z 705.901,A -85,B 0,C 180,E1 -6934.191,E2 -6934.191} C_VEL
LIN {X 0,Y 480.906,Z 702.34,A -85,B 0,C 180,E1 -6935.871,E2 -6935.871} C_VEL
LIN {X 0,Y 481.003,Z 697.469,A -85,B 0,C 180,E1 -6937.556,E2 -6937.556} C_VEL
LIN {X 0,Y 481.196,Z 691.162,A -85,B 0,C 180,E1 -6939.244,E2 -6939.244} C_VEL
LIN {X 0,Y 481.586,Z 683.251,A -85,B 0,C 180,E1 -6940.936,E2 -6940.936} C_VEL
LIN {X 0,Y 481.862,Z 675.32,A -85,B 0,C 180,E1 -6942.344,E2 -6942.344} C_VEL
LIN {X 0,Y 482.45,Z 664.703,A -85,B 0,C 180,E1 -6943.907,E2 -6943.907} C_VEL
LIN {X 0,Y 483.011,Z 654.359,A -85,B 0,C 180,E1 -6945.183,E2 -6945.183} C_VEL
LIN {X 0,Y 483.662,Z 643.249,A -85,B 0,C 180,E1 -6946.338,E2 -6946.338} C_VEL
LIN {X 0,Y 484.411,Z 630.983,A -85,B 0,C 180,E1 -6947.411,E2 -6947.411} C_VEL
LIN {X 0,Y 485.164,Z 617.838,A -85,B 0,C 180,E1 -6948.364,E2 -6948.364} C_VEL
LIN {X 0,Y 485.779,Z 605.415,A -85,B 0,C 180,E1 -6949.106,E2 -6949.106} C_VEL
LIN {X 0,Y 486.46,Z 591.432,A -85,B 0,C 180,E1 -6949.774,E2 -6949.774} C_VEL
LIN {X 0,Y 486.952,Z 576.604,A -85,B 0,C 180,E1 -6950.312,E2 -6950.312} C_VEL
LIN {X 0,Y 483.448,Z 560.857,A -85,B 0,C 180,E1 -6950.872,E2 -6950.872} C_VEL
LIN {X 0,Y 481.505,Z 552.065,A -85,B 0,C 180,E1 -6951.133,E2 -6951.133} C_VEL
LIN {X 0,Y 481.693,Z 543.694,A -85,B 0,C 180,E1 -6954.111,E2 -6954.111} C_VEL
LIN {X 0,Y 481.938,Z 535.304,A -85,B 0,C 180,E1 -6957.183,E2 -6957.183} C_VEL
LIN {X 0,Y 482.231,Z 527.329,A -85,B 0,C 180,E1 -6960.184,E2 -6960.184} C_VEL
LIN {X 0,Y 482.523,Z 519.853,A -85,B 0,C 180,E1 -6963.105,E2 -6963.105} C_VEL
LIN {X 0,Y 482.8,Z 512.427,A -85,B 0,C 180,E1 -6966.124,E2 -6966.124} C_VEL
LIN {X 0,Y 483.116,Z 506.283,A -85,B 0,C 180,E1 -6968.72,E2 -6968.72} C_VEL
LIN {X 0,Y 483.422,Z 500.194,A -85,B 0,C 180,E1 -6971.411,E2 -6971.411} C_VEL
LIN {X 0,Y 482.972,Z 496.178,A -85,B 0,C 180,E1 -6973.316,E2 -6973.316} C_VEL
LIN {X 0,Y 481.942,Z 490.56,A -85,B 0,C 180,E1 -6976.158,E2 -6976.158} C_VEL
LIN {X 0,Y 481.692,Z 489.111,A -85,B 0,C 180,E1 -6977.004,E2 -6977.004} C_VEL
LIN {X 0,Y 481.705,Z 489.11,A -85,B 0,C 180,E1 -6980.063,E2 -6980.063} C_VEL
LIN {X 0,Y 481.624,Z 489.119,A -85,B 0,C 180,E1 -6983.375,E2 -6983.375} C_VEL
LIN {X 0,Y 481.7,Z 489.109,A -85,B 0,C 180,E1 -6986.33,E2 -6986.33} C_VEL
LIN {X 0,Y 481.649,Z 489.116,A -85,B 0,C 180,E1 -6989.415,E2 -6989.415} C_VEL
LIN {X 0,Y 481.693,Z 489.108,A -85,B 0,C 180,E1 -6992.168,E2 -6992.168} C_VEL
LIN {X 0,Y 481.708,Z 489.107,A -85,B 0,C 180,E1 -6994.97,E2 -6994.97} C_VEL
LIN {X 0,Y 481.64,Z 489.117,A -85,B 0,C 180,E1 -6997.705,E2 -6997.705} C_VEL
LIN {X 0,Y 481.698,Z 489.108,A -85,B 0,C 180,E1 -7000.393,E2 -7000.393} C_VEL
LIN {X 0,Y 481.682,Z 489.112,A -85,B 0,C 180,E1 -7003.034,E2 -7003.034} C_VEL
LIN {X 0,Y 481.679,Z 489.112,A -85,B 0,C 180,E1 -7005.639,E2 -7005.639} C_VEL
LIN {X 0,Y 481.785,Z 489.098,A -85,B 0,C 180,E1 -7008.216,E2 -7008.216} C_VEL
LIN {X 0,Y 481.754,Z 489.104,A -85,B 0,C 180,E1 -7011.612,E2 -7011.612} C_VEL
LIN {X 0,Y 481.813,Z 489.094,A -85,B 0,C 180,E1 -7014.14,E2 -7014.14} C_VEL
LIN {X 0,Y 481.92,Z 489.083,A -85,B 0,C 180,E1 -7017.493,E2 -7017.493} C_VEL
LIN {X 0,Y 481.93,Z 489.08,A -85,B 0,C 180,E1 -7020,E2 -7020} C_VEL
LIN {X 0,Y 481.921,Z 489.08,A -85,B 0,C 180,E1 -7022.508,E2 -7022.508} C_VEL
LIN {X 0,Y 481.823,Z 489.095,A -85,B 0,C 180,E1 -7025.861,E2 -7025.861} C_VEL
LIN {X 0,Y 481.754,Z 489.101,A -85,B 0,C 180,E1 -7028.389,E2 -7028.389} C_VEL
LIN {X 0,Y 481.743,Z 489.104,A -85,B 0,C 180,E1 -7031.785,E2 -7031.785} C_VEL
LIN {X 0,Y 481.733,Z 489.106,A -85,B 0,C 180,E1 -7035.225,E2 -7035.225} C_VEL
LIN {X 0,Y 481.704,Z 489.107,A -85,B 0,C 180,E1 -7038.722,E2 -7038.722} C_VEL
LIN {X 0,Y 481.639,Z 489.118,A -85,B 0,C 180,E1 -7041.395,E2 -7041.395} C_VEL
LIN {X 0,Y 481.669,Z 489.112,A -85,B 0,C 180,E1 -7044.114,E2 -7044.114} C_VEL
LIN {X 0,Y 481.745,Z 489.104,A -85,B 0,C 180,E1 -7047.142,E2 -7047.142} C_VEL
LIN {X 0,Y 481.681,Z 489.112,A -85,B 0,C 180,E1 -7049.741,E2 -7049.741} C_VEL
LIN {X 0,Y 481.667,Z 489.112,A -85,B 0,C 180,E1 -7052.675,E2 -7052.675} C_VEL
LIN {X 0,Y 481.638,Z 489.119,A -85,B 0,C 180,E1 -7055.71,E2 -7055.71} C_VEL
LIN {X 0,Y 481.718,Z 489.108,A -85,B 0,C 180,E1 -7059.356,E2 -7059.356} C_VEL
LIN {X 0,Y 481.672,Z 489.113,A -85,B 0,C 180,E1 -7062.159,E2 -7062.159} C_VEL
LIN {X 0,Y 481.657,Z 489.113,A -85,B 0,C 180,E1 -7064.458,E2 -7064.458} C_VEL
LIN {X 0,Y 481.686,Z 489.11,A -85,B 0,C 180,E1 -7066.847,E2 -7066.847} C_VEL
LIN {X 0,Y 481.691,Z 489.11,A -85,B 0,C 180,E1 -7070.062,E2 -7070.062} C_VEL
LIN {X 0,Y 481.628,Z 489.118,A -85,B 0,C 180,E1 -7073.255,E2 -7073.255} C_VEL
LIN {X 0,Y 481.709,Z 489.107,A -85,B 0,C 180,E1 -7076.331,E2 -7076.331} C_VEL
LIN {X 0,Y 481.652,Z 489.116,A -85,B 0,C 180,E1 -7079.418,E2 -7079.418} C_VEL
LIN {X 0,Y 481.704,Z 489.108,A -85,B 0,C 180,E1 -7082.169,E2 -7082.169} C_VEL
LIN {X 0,Y 481.721,Z 489.106,A -85,B 0,C 180,E1 -7084.971,E2 -7084.971} C_VEL
LIN {X 0,Y 481.641,Z 489.116,A -85,B 0,C 180,E1 -7087.994,E2 -7087.994} C_VEL
LIN {X 0,Y 480.973,Z 489.199,A -85,B 0,C 180,E1 -7088.692,E2 -7088.692} C_VEL
LIN {X 0,Y 478.144,Z 489.554,A -85,B 0,C 180,E1 -7089.826,E2 -7089.826} C_VEL
LIN {X 0,Y 475.759,Z 489.85,A -85,B 0,C 180,E1 -7090.741,E2 -7090.741} C_VEL
LIN {X 0,Y 474.74,Z 489.977,A -85,B 0,C 180,E1 -7091.446,E2 -7091.446} C_VEL
LIN {X 0,Y 474.659,Z 489.987,A -85,B 0,C 180,E1 -7091.685,E2 -7091.685} C_VEL
LIN {X 0,Y 474.704,Z 489.979,A -85,B 0,C 180,E1 -7094.545,E2 -7094.545} C_VEL
LIN {X 0,Y 474.709,Z 489.979,A -85,B 0,C 180,E1 -7098.038,E2 -7098.038} C_VEL
LIN {X 0,Y 474.716,Z 489.98,A -85,B 0,C 180,E1 -7101.487,E2 -7101.487} C_VEL
LIN {X 0,Y 474.784,Z 489.971,A -85,B 0,C 180,E1 -7104.053,E2 -7104.053} C_VEL
LIN {X 0,Y 474.9,Z 489.957,A -85,B 0,C 180,E1 -7107.456,E2 -7107.456} C_VEL
LIN {X 0,Y 474.918,Z 489.954,A -85,B 0,C 180,E1 -7110,E2 -7110} C_VEL
LIN {X 0,Y 474.684,Z 489.982,A -85,B 0,C 180,E1 -7112.546,E2 -7112.546} C_VEL
LIN {X 0,Y 474.433,Z 490.016,A -85,B 0,C 180,E1 -7115.1,E2 -7115.1} C_VEL
LIN {X 0,Y 474.229,Z 490.042,A -85,B 0,C 180,E1 -7115.955,E2 -7115.955} C_VEL
LIN {X 0,Y 474.189,Z 492.204,A -85,B 0,C 180,E1 -7118.524,E2 -7118.524} C_VEL
LIN {X 0,Y 474.129,Z 495.314,A -85,B 0,C 180,E1 -7121.977,E2 -7121.977} C_VEL
LIN {X 0,Y 474.017,Z 498.516,A -85,B 0,C 180,E1 -7125.479,E2 -7125.479} C_VEL
LIN {X 0,Y 473.975,Z 501.416,A -85,B 0,C 180,E1 -7128.626,E2 -7128.626} C_VEL
LIN {X 0,Y 479.382,Z 518.867,A -85,B 0,C 180,E1 -7129.316,E2 -7129.316} C_VEL
LIN {X 0,Y 480.493,Z 524.275,A -85,B 0,C 180,E1 -7129.541,E2 -7129.541} C_VEL
LIN {X 0,Y 479.933,Z 539.66,A -85,B 0,C 180,E1 -7130.15,E2 -7130.15} C_VEL
LIN {X 0,Y 479.302,Z 552.845,A -85,B 0,C 180,E1 -7130.829,E2 -7130.829} C_VEL
LIN {X 0,Y 478.534,Z 566.589,A -85,B 0,C 180,E1 -7131.716,E2 -7131.716} C_VEL
LIN {X 0,Y 477.808,Z 579.136,A -85,B 0,C 180,E1 -7132.712,E2 -7132.712} C_VEL
LIN {X 0,Y 476.948,Z 591.278,A -85,B 0,C 180,E1 -7133.869,E2 -7133.869} C_VEL
LIN {X 0,Y 476.24,Z 602.091,A -85,B 0,C 180,E1 -7135.105,E2 -7135.105} C_VEL
LIN {X 0,Y 475.648,Z 611.081,A -85,B 0,C 180,E1 -7136.313,E2 -7136.313} C_VEL
LIN {X 0,Y 475.057,Z 620.515,A -85,B 0,C 180,E1 -7137.813,E2 -7137.813} C_VEL
LIN {X 0,Y 474.572,Z 629.234,A -85,B 0,C 180,E1 -7139.499,E2 -7139.499} C_VEL
LIN {X 0,Y 474.19,Z 636.536,A -85,B 0,C 180,E1 -7141.247,E2 -7141.247} C_VEL
LIN {X 0,Y 473.966,Z 641.627,A -85,B 0,C 180,E1 -7142.766,E2 -7142.766} C_VEL
LIN {X 0,Y 473.821,Z 645.704,A -85,B 0,C 180,E1 -7144.308,E2 -7144.308} C_VEL
LIN {X 0,Y 473.741,Z 647.871,A -85,B 0,C 180,E1 -7145.35,E2 -7145.35} C_VEL
LIN {X 0,Y 473.625,Z 650.03,A -85,B 0,C 180,E1 -7146.746,E2 -7146.746} C_VEL
LIN {X 0,Y 473.617,Z 651.723,A -85,B 0,C 180,E1 -7148.553,E2 -7148.553} C_VEL
LIN {X 0,Y 473.58,Z 652.137,A -85,B 0,C 180,E1 -7149.652,E2 -7149.652} C_VEL
LIN {X 0,Y 473.614,Z 652.077,A -85,B 0,C 180,E1 -7150.817,E2 -7150.817} C_VEL
LIN {X 0,Y 473.621,Z 651.389,A -85,B 0,C 180,E1 -7152.102,E2 -7152.102} C_VEL
LIN {X 0,Y 473.699,Z 650.058,A -85,B 0,C 180,E1 -7153.365,E2 -7153.365} C_VEL
LIN {X 0,Y 473.76,Z 648.19,A -85,B 0,C 180,E1 -7154.597,E2 -7154.597} C_VEL
LIN {X 0,Y 473.864,Z 645.735,A -85,B 0,C 180,E1 -7155.807,E2 -7155.807} C_VEL
LIN {X 0,Y 474.038,Z 641.385,A -85,B 0,C 180,E1 -7157.451,E2 -7157.451} C_VEL
LIN {X 0,Y 474.257,Z 634.986,A -85,B 0,C 180,E1 -7159.304,E2 -7159.304} C_VEL
LIN {X 0,Y 474.707,Z 627.499,A -85,B 0,C 180,E1 -7161.008,E2 -7161.008} C_VEL
LIN {X 0,Y 475.232,Z 618.458,A -85,B 0,C 180,E1 -7162.675,E2 -7162.675} C_VEL
LIN {X 0,Y 475.814,Z 609.256,A -85,B 0,C 180,E1 -7164.085,E2 -7164.085} C_VEL
LIN {X 0,Y 476.601,Z 597.972,A -85,B 0,C 180,E1 -7165.52,E2 -7165.52} C_VEL
LIN {X 0,Y 477.372,Z 586.452,A -85,B 0,C 180,E1 -7166.742,E2 -7166.742} C_VEL
LIN {X 0,Y 478.106,Z 574.506,A -85,B 0,C 180,E1 -7167.8,E2 -7167.8} C_VEL
LIN {X 0,Y 478.95,Z 561.212,A -85,B 0,C 180,E1 -7168.769,E2 -7168.769} C_VEL
LIN {X 0,Y 479.633,Z 547.513,A -85,B 0,C 180,E1 -7169.577,E2 -7169.577} C_VEL
LIN {X 0,Y 480.26,Z 532.49,A -85,B 0,C 180,E1 -7170.267,E2 -7170.267} C_VEL
LIN {X 0,Y 480.421,Z 523.128,A -85,B 0,C 180,E1 -7170.61,E2 -7170.61} C_VEL
LIN {X 0,Y 477.929,Z 513.963,A -85,B 0,C 180,E1 -7171,E2 -7171} C_VEL
LIN {X 0,Y 473.972,Z 502.269,A -85,B 0,C 180,E1 -7171.457,E2 -7171.457} C_VEL
LIN {X 0,Y 474.095,Z 499.45,A -85,B 0,C 180,E1 -7174.723,E2 -7174.723} C_VEL
LIN {X 0,Y 474.12,Z 497.256,A -85,B 0,C 180,E1 -7177.331,E2 -7177.331} C_VEL
LIN {X 0,Y 474.219,Z 494.978,A -85,B 0,C 180,E1 -7180.07,E2 -7180.07} C_VEL
LIN {X 0,Y 474.311,Z 492.727,A -85,B 0,C 180,E1 -7182.761,E2 -7182.761} C_VEL
LIN {X 0,Y 474.352,Z 490.532,A -85,B 0,C 180,E1 -7185.411,E2 -7185.411} C_VEL
LIN {X 0,Y 474.395,Z 490.022,A -85,B 0,C 180,E1 -7186.288,E2 -7186.288} C_VEL
LIN {X 0,Y 474.646,Z 489.987,A -85,B 0,C 180,E1 -7188.902,E2 -7188.902} C_VEL
LIN {X 0,Y 474.792,Z 489.969,A -85,B 0,C 180,E1 -7192.344,E2 -7192.344} C_VEL
LIN {X 0,Y 474.753,Z 489.971,A -85,B 0,C 180,E1 -7194.904,E2 -7194.904} C_VEL
LIN {X 0,Y 474.892,Z 489.957,A -85,B 0,C 180,E1 -7197.455,E2 -7197.455} C_VEL
LIN {X 0,Y 474.908,Z 489.954,A -85,B 0,C 180,E1 -7200,E2 -7200} C_VEL
LIN {X 0,Y 474.89,Z 489.953,A -85,B 0,C 180,E1 -7202.544,E2 -7202.544} C_VEL
LIN {X 0,Y 474.78,Z 489.968,A -85,B 0,C 180,E1 -7205.947,E2 -7205.947} C_VEL
LIN {X 0,Y 474.725,Z 489.975,A -85,B 0,C 180,E1 -7208.513,E2 -7208.513} C_VEL
LIN {X 0,Y 474.701,Z 489.976,A -85,B 0,C 180,E1 -7211.962,E2 -7211.962} C_VEL
LIN {X 0,Y 474.695,Z 489.977,A -85,B 0,C 180,E1 -7215.456,E2 -7215.456} C_VEL
LIN {X 0,Y 474.661,Z 489.983,A -85,B 0,C 180,E1 -7219.01,E2 -7219.01} C_VEL
LIN {X 0,Y 474.587,Z 489.99,A -85,B 0,C 180,E1 -7221.729,E2 -7221.729} C_VEL
LIN {X 0,Y 474.655,Z 489.986,A -85,B 0,C 180,E1 -7224.493,E2 -7224.493} C_VEL
LIN {X 0,Y 474.695,Z 489.978,A -85,B 0,C 180,E1 -7227.339,E2 -7227.339} C_VEL
LIN {X 0,Y 474.607,Z 489.99,A -85,B 0,C 180,E1 -7230.811,E2 -7230.811} C_VEL
LIN {X 0,Y 474.635,Z 489.99,A -85,B 0,C 180,E1 -7233.984,E2 -7233.984} C_VEL
LIN {X 0,Y 474.572,Z 489.996,A -85,B 0,C 180,E1 -7236.9,E2 -7236.9} C_VEL
LIN {X 0,Y 474.625,Z 489.986,A -85,B 0,C 180,E1 -7239.648,E2 -7239.648} C_VEL
LIN {X 0,Y 474.677,Z 490.172,A -85,B 0,C 180,E1 -7242.734,E2 -7242.734} C_VEL
LIN {X 0,Y 475.698,Z 495.87,A -85,B 0,C 180,E1 -7246.023,E2 -7246.023} C_VEL
LIN {X 0,Y 476.245,Z 500.432,A -85,B 0,C 180,E1 -7248.389,E2 -7248.389} C_VEL
LIN {X 0,Y 476.037,Z 505.142,A -85,B 0,C 180,E1 -7250.593,E2 -7250.593} C_VEL
LIN {X 0,Y 475.678,Z 512.301,A -85,B 0,C 180,E1 -7253.773,E2 -7253.773} C_VEL
LIN {X 0,Y 475.331,Z 519.683,A -85,B 0,C 180,E1 -7256.834,E2 -7256.834} C_VEL
LIN {X 0,Y 475.158,Z 525.336,A -85,B 0,C 180,E1 -7259.078,E2 -7259.078} C_VEL
LIN {X 0,Y 474.831,Z 533.506,A -85,B 0,C 180,E1 -7262.211,E2 -7262.211} C_VEL
LIN {X 0,Y 474.654,Z 539.902,A -85,B 0,C 180,E1 -7264.582,E2 -7264.582} C_VEL
LIN {X 0,Y 474.441,Z 548.854,A -85,B 0,C 180,E1 -7267.806,E2 -7267.806} C_VEL
LIN {X 0,Y 474.426,Z 550.95,A -85,B 0,C 180,E1 -7268.551,E2 -7268.551} C_VEL
LIN {X 0,Y 478.097,Z 568.188,A -85,B 0,C 180,E1 -7269.082,E2 -7269.082} C_VEL
LIN {X 0,Y 480.208,Z 578.308,A -85,B 0,C 180,E1 -7269.482,E2 -7269.482} C_VEL
LIN {X 0,Y 479.623,Z 591.781,A -85,B 0,C 180,E1 -7269.995,E2 -7269.995} C_VEL
LIN {X 0,Y 478.883,Z 606.376,A -85,B 0,C 180,E1 -7270.719,E2 -7270.719} C_VEL
LIN {X 0,Y 478.127,Z 620.051,A -85,B 0,C 180,E1 -7271.577,E2 -7271.577} C_VEL
LIN {X 0,Y 477.267,Z 633.977,A -85,B 0,C 180,E1 -7272.651,E2 -7272.651} C_VEL
LIN {X 0,Y 476.514,Z 646.6,A -85,B 0,C 180,E1 -7273.836,E2 -7273.836} C_VEL
LIN {X 0,Y 475.832,Z 657.193,A -85,B 0,C 180,E1 -7275.02,E2 -7275.02} C_VEL
LIN {X 0,Y 475.272,Z 667.034,A -85,B 0,C 180,E1 -7276.314,E2 -7276.314} C_VEL
LIN {X 0,Y 474.71,Z 676.11,A -85,B 0,C 180,E1 -7277.719,E2 -7277.719} C_VEL
LIN {X 0,Y 474.483,Z 683.745,A -85,B 0,C 180,E1 -7279.114,E2 -7279.114} C_VEL
LIN {X 0,Y 474.105,Z 690.589,A -85,B 0,C 180,E1 -7280.615,E2 -7280.615} C_VEL
LIN {X 0,Y 473.925,Z 696.928,A -85,B 0,C 180,E1 -7282.33,E2 -7282.33} C_VEL
LIN {X 0,Y 473.815,Z 701.833,A -85,B 0,C 180,E1 -7284.04,E2 -7284.04} C_VEL
LIN {X 0,Y 473.712,Z 705.426,A -85,B 0,C 180,E1 -7285.746,E2 -7285.746} C_VEL
LIN {X 0,Y 473.797,Z 706.768,A -85,B 0,C 180,E1 -7286.598,E2 -7286.598} C_VEL
LIN {X 0,Y 473.747,Z 708.546,A -85,B 0,C 180,E1 -7288.299,E2 -7288.299} C_VEL
LIN {X 0,Y 473.666,Z 709.158,A -85,B 0,C 180,E1 -7290,E2 -7290} C_VEL
LIN {X 0,Y 473.747,Z 708.564,A -85,B 0,C 180,E1 -7291.7,E2 -7291.7} C_VEL
LIN {X 0,Y 473.797,Z 706.806,A -85,B 0,C 180,E1 -7293.401,E2 -7293.401} C_VEL
LIN {X 0,Y 473.788,Z 703.856,A -85,B 0,C 180,E1 -7295.106,E2 -7295.106} C_VEL
LIN {X 0,Y 473.885,Z 699.653,A -85,B 0,C 180,E1 -7296.813,E2 -7296.813} C_VEL
LIN {X 0,Y 474.032,Z 694.08,A -85,B 0,C 180,E1 -7298.526,E2 -7298.526} C_VEL
LIN {X 0,Y 474.273,Z 686.991,A -85,B 0,C 180,E1 -7300.242,E2 -7300.242} C_VEL
LIN {X 0,Y 474.636,Z 679.415,A -85,B 0,C 180,E1 -7301.747,E2 -7301.747} C_VEL
LIN {X 0,Y 475.088,Z 670.284,A -85,B 0,C 180,E1 -7303.255,E2 -7303.255} C_VEL
LIN {X 0,Y 475.748,Z 659.316,A -85,B 0,C 180,E1 -7304.763,E2 -7304.763} C_VEL
LIN {X 0,Y 476.497,Z 648.041,A -85,B 0,C 180,E1 -7306.054,E2 -7306.054} C_VEL
LIN {X 0,Y 477.221,Z 635.69,A -85,B 0,C 180,E1 -7307.239,E2 -7307.239} C_VEL
LIN {X 0,Y 478.155,Z 622.131,A -85,B 0,C 180,E1 -7308.31,E2 -7308.31} C_VEL
LIN {X 0,Y 478.802,Z 608.817,A -85,B 0,C 180,E1 -7309.173,E2 -7309.173} C_VEL
LIN {X 0,Y 479.6,Z 594.16,A -85,B 0,C 180,E1 -7309.925,E2 -7309.925} C_VEL
LIN {X 0,Y 480.222,Z 578.845,A -85,B 0,C 180,E1 -7310.522,E2 -7310.522} C_VEL
LIN {X 0,Y 479.432,Z 573.977,A -85,B 0,C 180,E1 -7310.71,E2 -7310.71} C_VEL
LIN {X 0,Y 475.836,Z 557.974,A -85,B 0,C 180,E1 -7311.267,E2 -7311.267} C_VEL
LIN {X 0,Y 474.459,Z 551.694,A -85,B 0,C 180,E1 -7311.448,E2 -7311.448} C_VEL
LIN {X 0,Y 474.666,Z 543.377,A -85,B 0,C 180,E1 -7314.491,E2 -7314.491} C_VEL
LIN {X 0,Y 474.913,Z 535.584,A -85,B 0,C 180,E1 -7317.389,E2 -7317.389} C_VEL
LIN {X 0,Y 475.203,Z 528.259,A -85,B 0,C 180,E1 -7320.187,E2 -7320.187} C_VEL
LIN {X 0,Y 475.529,Z 520.826,A -85,B 0,C 180,E1 -7323.149,E2 -7323.149} C_VEL
LIN {X 0,Y 475.818,Z 513.414,A -85,B 0,C 180,E1 -7326.213,E2 -7326.213} C_VEL
LIN {X 0,Y 476.243,Z 506.048,A -85,B 0,C 180,E1 -7329.386,E2 -7329.386} C_VEL
LIN {X 0,Y 476.43,Z 501.173,A -85,B 0,C 180,E1 -7331.59,E2 -7331.59} C_VEL
LIN {X 0,Y 475.806,Z 496.299,A -85,B 0,C 180,E1 -7333.964,E2 -7333.964} C_VEL
LIN {X 0,Y 474.675,Z 489.985,A -85,B 0,C 180,E1 -7337.36,E2 -7337.36} C_VEL
LIN {X 0,Y 474.675,Z 489.985,A -85,B 0,C 180,E1 -7340.457,E2 -7340.457} C_VEL
LIN {X 0,Y 474.585,Z 489.995,A -85,B 0,C 180,E1 -7343.676,E2 -7343.676} C_VEL
LIN {X 0,Y 474.634,Z 489.989,A -85,B 0,C 180,E1 -7346.78,E2 -7346.78} C_VEL
LIN {X 0,Y 474.605,Z 489.994,A -85,B 0,C 180,E1 -7349.77,E2 -7349.77} C_VEL
LIN {X 0,Y 474.705,Z 489.978,A -85,B 0,C 180,E1 -7352.681,E2 -7352.681} C_VEL
LIN {X 0,Y 474.649,Z 489.988,A -85,B 0,C 180,E1 -7355.507,E2 -7355.507} C_VEL
LIN {X 0,Y 474.66,Z 489.986,A -85,B 0,C 180,E1 -7359.185,E2 -7359.185} C_VEL
LIN {X 0,Y 474.647,Z 489.988,A -85,B 0,C 180,E1 -7361.884,E2 -7361.884} C_VEL
LIN {X 0,Y 474.689,Z 489.98,A -85,B 0,C 180,E1 -7364.544,E2 -7364.544} C_VEL
LIN {X 0,Y 474.729,Z 489.978,A -85,B 0,C 180,E1 -7368.039,E2 -7368.039} C_VEL
LIN {X 0,Y 474.719,Z 489.979,A -85,B 0,C 180,E1 -7371.487,E2 -7371.487} C_VEL
LIN {X 0,Y 474.774,Z 489.971,A -85,B 0,C 180,E1 -7374.053,E2 -7374.053} C_VEL
LIN {X 0,Y 474.886,Z 489.959,A -85,B 0,C 180,E1 -7377.456,E2 -7377.456} C_VEL
LIN {X 0,Y 474.867,Z 489.96,A -85,B 0,C 180,E1 -7380.848,E2 -7380.848} C_VEL
LIN {X 0,Y 474.887,Z 489.956,A -85,B 0,C 180,E1 -7382.545,E2 -7382.545} C_VEL
LIN {X 0,Y 474.783,Z 489.971,A -85,B 0,C 180,E1 -7385.948,E2 -7385.948} C_VEL
LIN {X 0,Y 474.719,Z 489.977,A -85,B 0,C 180,E1 -7388.514,E2 -7388.514} C_VEL
LIN {X 0,Y 474.696,Z 489.981,A -85,B 0,C 180,E1 -7391.963,E2 -7391.963} C_VEL
LIN {X 0,Y 474.69,Z 489.983,A -85,B 0,C 180,E1 -7395.456,E2 -7395.456} C_VEL
LIN {X 0,Y 474.657,Z 489.985,A -85,B 0,C 180,E1 -7399.011,E2 -7399.011} C_VEL
LIN {X 0,Y 474.582,Z 489.996,A -85,B 0,C 180,E1 -7401.73,E2 -7401.73} C_VEL
LIN {X 0,Y 474.651,Z 489.985,A -85,B 0,C 180,E1 -7404.494,E2 -7404.494} C_VEL
LIN {X 0,Y 474.692,Z 489.983,A -85,B 0,C 180,E1 -7407.34,E2 -7407.34} C_VEL
LIN {X 0,Y 474.603,Z 489.992,A -85,B 0,C 180,E1 -7410.812,E2 -7410.812} C_VEL
LIN {X 0,Y 474.632,Z 489.989,A -85,B 0,C 180,E1 -7413.985,E2 -7413.985} C_VEL
LIN {X 0,Y 474.571,Z 489.996,A -85,B 0,C 180,E1 -7416.901,E2 -7416.901} C_VEL
LIN {X 0,Y 474.662,Z 489.986,A -85,B 0,C 180,E1 -7419.655,E2 -7419.655} C_VEL
LIN {X 0,Y 474.649,Z 489.987,A -85,B 0,C 180,E1 -7422.931,E2 -7422.931} C_VEL
LIN {X 0,Y 474.615,Z 489.992,A -85,B 0,C 180,E1 -7425.897,E2 -7425.897} C_VEL
LIN {X 0,Y 474.644,Z 489.987,A -85,B 0,C 180,E1 -7429.039,E2 -7429.039} C_VEL
LIN {X 0,Y 474.618,Z 489.992,A -85,B 0,C 180,E1 -7431.704,E2 -7431.704} C_VEL
LIN {X 0,Y 474.629,Z 489.989,A -85,B 0,C 180,E1 -7434.727,E2 -7434.727} C_VEL
LIN {X 0,Y 474.637,Z 489.99,A -85,B 0,C 180,E1 -7437.789,E2 -7437.789} C_VEL
LIN {X 0,Y 474.625,Z 489.988,A -85,B 0,C 180,E1 -7440.886,E2 -7440.886} C_VEL
LIN {X 0,Y 474.669,Z 489.986,A -85,B 0,C 180,E1 -7443.63,E2 -7443.63} C_VEL
LIN {X 0,Y 474.638,Z 489.987,A -85,B 0,C 180,E1 -7446.642,E2 -7446.642} C_VEL
LIN {X 0,Y 474.658,Z 489.985,A -85,B 0,C 180,E1 -7450.091,E2 -7450.091} C_VEL
LIN {X 0,Y 474.659,Z 489.987,A -85,B 0,C 180,E1 -7451.685,E2 -7451.685} C_VEL
LIN {X 0,Y 473.997,Z 490.07,A -85,B 0,C 180,E1 -7452.394,E2 -7452.394} C_VEL
LIN {X 0,Y 471.146,Z 490.426,A -85,B 0,C 180,E1 -7453.546,E2 -7453.546} C_VEL
LIN {X 0,Y 468.729,Z 490.726,A -85,B 0,C 180,E1 -7454.474,E2 -7454.474} C_VEL
LIN {X 0,Y 467.687,Z 490.854,A -85,B 0,C 180,E1 -7455.191,E2 -7455.191} C_VEL
LIN {X 0,Y 467.601,Z 490.864,A -85,B 0,C 180,E1 -7455.434,E2 -7455.434} C_VEL
LIN {X 0,Y 467.656,Z 490.857,A -85,B 0,C 180,E1 -7458.735,E2 -7458.735} C_VEL
LIN {X 0,Y 467.674,Z 490.857,A -85,B 0,C 180,E1 -7461.358,E2 -7461.358} C_VEL
LIN {X 0,Y 467.748,Z 490.848,A -85,B 0,C 180,E1 -7463.963,E2 -7463.963} C_VEL
LIN {X 0,Y 467.865,Z 490.833,A -85,B 0,C 180,E1 -7467.418,E2 -7467.418} C_VEL
LIN {X 0,Y 467.888,Z 490.829,A -85,B 0,C 180,E1 -7470,E2 -7470} C_VEL
LIN {X 0,Y 467.638,Z 490.859,A -85,B 0,C 180,E1 -7472.585,E2 -7472.585} C_VEL
LIN {X 0,Y 467.362,Z 490.897,A -85,B 0,C 180,E1 -7475.177,E2 -7475.177} C_VEL
LIN {X 0,Y 467.175,Z 490.92,A -85,B 0,C 180,E1 -7476.045,E2 -7476.045} C_VEL
LIN {X 0,Y 467.132,Z 493.035,A -85,B 0,C 180,E1 -7478.653,E2 -7478.653} C_VEL
LIN {X 0,Y 467.038,Z 496.194,A -85,B 0,C 180,E1 -7482.162,E2 -7482.162} C_VEL
LIN {X 0,Y 466.962,Z 498.584,A -85,B 0,C 180,E1 -7484.825,E2 -7484.825} C_VEL
LIN {X 0,Y 466.888,Z 501.784,A -85,B 0,C 180,E1 -7488.286,E2 -7488.286} C_VEL
LIN {X 0,Y 472.683,Z 520.016,A -85,B 0,C 180,E1 -7489.037,E2 -7489.037} C_VEL
LIN {X 0,Y 473.799,Z 525.439,A -85,B 0,C 180,E1 -7489.271,E2 -7489.271} C_VEL
LIN {X 0,Y 473.272,Z 539.962,A -85,B 0,C 180,E1 -7489.858,E2 -7489.858} C_VEL
LIN {X 0,Y 472.533,Z 554.73,A -85,B 0,C 180,E1 -7490.642,E2 -7490.642} C_VEL
LIN {X 0,Y 471.726,Z 567.971,A -85,B 0,C 180,E1 -7491.523,E2 -7491.523} C_VEL
LIN {X 0,Y 470.97,Z 580.328,A -85,B 0,C 180,E1 -7492.528,E2 -7492.528} C_VEL
LIN {X 0,Y 470.072,Z 592.254,A -85,B 0,C 180,E1 -7493.691,E2 -7493.691} C_VEL
LIN {X 0,Y 469.292,Z 603.652,A -85,B 0,C 180,E1 -7495.028,E2 -7495.028} C_VEL
LIN {X 0,Y 468.572,Z 614.211,A -85,B 0,C 180,E1 -7496.515,E2 -7496.515} C_VEL
LIN {X 0,Y 467.971,Z 622.92,A -85,B 0,C 180,E1 -7497.99,E2 -7497.99} C_VEL
LIN {X 0,Y 467.47,Z 631.482,A -85,B 0,C 180,E1 -7499.744,E2 -7499.744} C_VEL
LIN {X 0,Y 467.137,Z 637.743,A -85,B 0,C 180,E1 -7501.334,E2 -7501.334} C_VEL
LIN {X 0,Y 466.906,Z 642.472,A -85,B 0,C 180,E1 -7502.812,E2 -7502.812} C_VEL
LIN {X 0,Y 466.788,Z 645.812,A -85,B 0,C 180,E1 -7504.097,E2 -7504.097} C_VEL
LIN {X 0,Y 466.582,Z 649.445,A -85,B 0,C 180,E1 -7505.976,E2 -7505.976} C_VEL
LIN {X 0,Y 466.548,Z 650.911,A -85,B 0,C 180,E1 -7507.053,E2 -7507.053} C_VEL
LIN {X 0,Y 466.545,Z 652.092,A -85,B 0,C 180,E1 -7508.433,E2 -7508.433} C_VEL
